LIN {X 0,Y 187.454,Z 298.954,A -85,B 0,C 180,E1 -22168.909,E2 -22168.909} C_VEL
LIN {X 0,Y 190.093,Z 301.065,A -85,B 0,C 180,E1 -22170.478,E2 -22170.478} C_VEL
LIN {X 0,Y 192.091,Z 304.274,A -85,B 0,C 180,E1 -22171.704,E2 -22171.704} C_VEL
LIN {X 0,Y 194.183,Z 306.294,A -85,B 0,C 180,E1 -22172.829,E2 -22172.829} C_VEL
LIN {X 0,Y 196.909,Z 310.048,A -85,B 0,C 180,E1 -22174.282,E2 -22174.282} C_VEL
LIN {X 0,Y 198.155,Z 311.601,A -85,B 0,C 180,E1 -22174.905,E2 -22174.905} C_VEL
LIN {X 0,Y 202.245,Z 317.198,A -85,B 0,C 180,E1 -22176.865,E2 -22176.865} C_VEL
LIN {X 0,Y 207.451,Z 324.554,A -85,B 0,C 180,E1 -22179.145,E2 -22179.145} C_VEL
LIN {X 0,Y 212.469,Z 332.432,A -85,B 0,C 180,E1 -22181.182,E2 -22181.182} C_VEL
LIN {X 0,Y 218.995,Z 345.187,A -85,B 0,C 180,E1 -22183.701,E2 -22183.701} C_VEL
LIN {X 0,Y 224.024,Z 356.545,A -85,B 0,C 180,E1 -22185.537,E2 -22185.537} C_VEL
LIN {X 0,Y 225.79,Z 360.908,A -85,B 0,C 180,E1 -22186.166,E2 -22186.166} C_VEL
LIN {X 0,Y 221.73,Z 427.354,A -85,B 0,C 180,E1 -22188.125,E2 -22188.125} C_VEL
LIN {X 0,Y 219.881,Z 441.769,A -85,B 0,C 180,E1 -22188.836,E2 -22188.836} C_VEL
LIN {X 0,Y 217.42,Z 455.664,A -85,B 0,C 180,E1 -22189.875,E2 -22189.875} C_VEL
LIN {X 0,Y 214.477,Z 468.601,A -85,B 0,C 180,E1 -22191.195,E2 -22191.195} C_VEL
LIN {X 0,Y 211.037,Z 481.143,A -85,B 0,C 180,E1 -22192.872,E2 -22192.872} C_VEL
LIN {X 0,Y 207.458,Z 492.576,A -85,B 0,C 180,E1 -22194.838,E2 -22194.838} C_VEL
LIN {X 0,Y 203.569,Z 503.074,A -85,B 0,C 180,E1 -22197.061,E2 -22197.061} C_VEL
LIN {X 0,Y 199.991,Z 511.877,A -85,B 0,C 180,E1 -22199.367,E2 -22199.367} C_VEL
LIN {X 0,Y 196.158,Z 520.748,A -85,B 0,C 180,E1 -22202.241,E2 -22202.241} C_VEL
LIN {X 0,Y 192.263,Z 529.243,A -85,B 0,C 180,E1 -22205.718,E2 -22205.718} C_VEL
LIN {X 0,Y 189.302,Z 536.081,A -85,B 0,C 180,E1 -22209.348,E2 -22209.348} C_VEL
LIN {X 0,Y 187.05,Z 540.801,A -85,B 0,C 180,E1 -22212.508,E2 -22212.508} C_VEL
LIN {X 0,Y 184.934,Z 545.689,A -85,B 0,C 180,E1 -22216.82,E2 -22216.82} C_VEL
LIN {X 0,Y 183.7,Z 549.087,A -85,B 0,C 180,E1 -22221.197,E2 -22221.197} C_VEL
LIN {X 0,Y 183.124,Z 551.102,A -85,B 0,C 180,E1 -22225.598,E2 -22225.598} C_VEL
LIN {X 0,Y 183.07,Z 551.787,A -85,B 0,C 180,E1 -22230,E2 -22230} C_VEL
LIN {X 0,Y 183.124,Z 551.153,A -85,B 0,C 180,E1 -22234.402,E2 -22234.402} C_VEL
LIN {X 0,Y 183.693,Z 549.184,A -85,B 0,C 180,E1 -22238.803,E2 -22238.803} C_VEL
LIN {X 0,Y 184.898,Z 545.833,A -85,B 0,C 180,E1 -22243.182,E2 -22243.182} C_VEL
LIN {X 0,Y 187.018,Z 540.999,A -85,B 0,C 180,E1 -22247.495,E2 -22247.495} C_VEL
LIN {X 0,Y 189.204,Z 536.332,A -85,B 0,C 180,E1 -22250.663,E2 -22250.663} C_VEL
LIN {X 0,Y 192.218,Z 529.549,A -85,B 0,C 180,E1 -22254.288,E2 -22254.288} C_VEL
LIN {X 0,Y 196.084,Z 521.119,A -85,B 0,C 180,E1 -22257.77,E2 -22257.77} C_VEL
LIN {X 0,Y 199.918,Z 512.321,A -85,B 0,C 180,E1 -22260.645,E2 -22260.645} C_VEL
LIN {X 0,Y 203.47,Z 503.606,A -85,B 0,C 180,E1 -22262.956,E2 -22262.956} C_VEL
LIN {X 0,Y 207.368,Z 493.216,A -85,B 0,C 180,E1 -22265.179,E2 -22265.179} C_VEL
LIN {X 0,Y 210.969,Z 481.914,A -85,B 0,C 180,E1 -22267.141,E2 -22267.141} C_VEL
LIN {X 0,Y 214.39,Z 469.557,A -85,B 0,C 180,E1 -22268.824,E2 -22268.824} C_VEL
LIN {X 0,Y 217.582,Z 455.768,A -85,B 0,C 180,E1 -22270.24,E2 -22270.24} C_VEL
LIN {X 0,Y 220.064,Z 441.904,A -85,B 0,C 180,E1 -22271.274,E2 -22271.274} C_VEL
LIN {X 0,Y 221.841,Z 427.094,A -85,B 0,C 180,E1 -22272.032,E2 -22272.032} C_VEL
LIN {X 0,Y 224.773,Z 380.963,A -85,B 0,C 180,E1 -22273.381,E2 -22273.381} C_VEL
LIN {X 0,Y 225.874,Z 360.793,A -85,B 0,C 180,E1 -22273.985,E2 -22273.985} C_VEL
LIN {X 0,Y 219.562,Z 346.139,A -85,B 0,C 180,E1 -22276.275,E2 -22276.275} C_VEL
LIN {X 0,Y 213.002,Z 333.315,A -85,B 0,C 180,E1 -22278.794,E2 -22278.794} C_VEL
LIN {X 0,Y 208.872,Z 326.562,A -85,B 0,C 180,E1 -22280.464,E2 -22280.464} C_VEL
LIN {X 0,Y 203.086,Z 318.318,A -85,B 0,C 180,E1 -22282.96,E2 -22282.96} C_VEL
LIN {X 0,Y 200.505,Z 314.745,A -85,B 0,C 180,E1 -22284.165,E2 -22284.165} C_VEL
LIN {X 0,Y 197.121,Z 310.237,A -85,B 0,C 180,E1 -22285.838,E2 -22285.838} C_VEL
LIN {X 0,Y 194.35,Z 306.597,A -85,B 0,C 180,E1 -22287.306,E2 -22287.306} C_VEL
LIN {X 0,Y 193.477,Z 305.537,A -85,B 0,C 180,E1 -22287.784,E2 -22287.784} C_VEL
LIN {X 0,Y 191.048,Z 302.837,A -85,B 0,C 180,E1 -22289.155,E2 -22289.155} C_VEL
LIN {X 0,Y 189.729,Z 300.609,A -85,B 0,C 180,E1 -22289.995,E2 -22289.995} C_VEL
LIN {X 0,Y 187.251,Z 298.716,A -85,B 0,C 180,E1 -22291.486,E2 -22291.486} C_VEL
LIN {X 0,Y 185.658,Z 295.648,A -85,B 0,C 180,E1 -22292.831,E2 -22292.831} C_VEL
LIN {X 0,Y 185.553,Z 295.014,A -85,B 0,C 180,E1 -22293.574,E2 -22293.574} C_VEL
LIN {X 0,Y 185.593,Z 294.976,A -85,B 0,C 180,E1 -22297.748,E2 -22297.748} C_VEL
LIN {X 0,Y 185.686,Z 294.979,A -85,B 0,C 180,E1 -22302.375,E2 -22302.375} C_VEL
LIN {X 0,Y 185.727,Z 294.959,A -85,B 0,C 180,E1 -22306.877,E2 -22306.877} C_VEL
LIN {X 0,Y 185.979,Z 294.915,A -85,B 0,C 180,E1 -22311.306,E2 -22311.306} C_VEL
LIN {X 0,Y 186.202,Z 294.886,A -85,B 0,C 180,E1 -22317.837,E2 -22317.837} C_VEL
LIN {X 0,Y 186.405,Z 294.881,A -85,B 0,C 180,E1 -22320,E2 -22320} C_VEL
LIN {X 0,Y 185.919,Z 294.922,A -85,B 0,C 180,E1 -22324.336,E2 -22324.336} C_VEL
LIN {X 0,Y 186.01,Z 294.921,A -85,B 0,C 180,E1 -22328.692,E2 -22328.692} C_VEL
LIN {X 0,Y 185.76,Z 294.97,A -85,B 0,C 180,E1 -22333.121,E2 -22333.121} C_VEL
LIN {X 0,Y 185.691,Z 294.975,A -85,B 0,C 180,E1 -22338.884,E2 -22338.884} C_VEL
LIN {X 0,Y 185.598,Z 294.99,A -85,B 0,C 180,E1 -22344.663,E2 -22344.663} C_VEL
LIN {X 0,Y 185.575,Z 295.249,A -85,B 0,C 180,E1 -22346.726,E2 -22346.726} C_VEL
LIN {X 0,Y 185.908,Z 296.393,A -85,B 0,C 180,E1 -22347.434,E2 -22347.434} C_VEL
LIN {X 0,Y 187.453,Z 298.923,A -85,B 0,C 180,E1 -22348.556,E2 -22348.556} C_VEL
LIN {X 0,Y 190.034,Z 300.979,A -85,B 0,C 180,E1 -22350.104,E2 -22350.104} C_VEL
LIN {X 0,Y 192.02,Z 304.151,A -85,B 0,C 180,E1 -22351.334,E2 -22351.334} C_VEL
LIN {X 0,Y 194.193,Z 306.346,A -85,B 0,C 180,E1 -22352.518,E2 -22352.518} C_VEL
LIN {X 0,Y 196.687,Z 309.82,A -85,B 0,C 180,E1 -22353.862,E2 -22353.862} C_VEL
LIN {X 0,Y 198.125,Z 311.496,A -85,B 0,C 180,E1 -22354.58,E2 -22354.58} C_VEL
LIN {X 0,Y 201.006,Z 315.29,A -85,B 0,C 180,E1 -22355.979,E2 -22355.979} C_VEL
LIN {X 0,Y 204.724,Z 320.809,A -85,B 0,C 180,E1 -22357.697,E2 -22357.697} C_VEL
LIN {X 0,Y 210.721,Z 330.915,A -85,B 0,C 180,E1 -22360.281,E2 -22360.281} C_VEL
LIN {X 0,Y 216.173,Z 341.306,A -85,B 0,C 180,E1 -22362.457,E2 -22362.457} C_VEL
LIN {X 0,Y 221.573,Z 352.961,A -85,B 0,C 180,E1 -22364.49,E2 -22364.49} C_VEL
LIN {X 0,Y 225.817,Z 363.464,A -85,B 0,C 180,E1 -22366.03,E2 -22366.03} C_VEL
LIN {X 0,Y 225.111,Z 375.8,A -85,B 0,C 180,E1 -22366.391,E2 -22366.391} C_VEL
LIN {X 0,Y 224.205,Z 381.65,A -85,B 0,C 180,E1 -22366.424,E2 -22366.424} C_VEL
LIN {X 0,Y 218.939,Z 400.687,A -85,B 0,C 180,E1 -22365.957,E2 -22365.957} C_VEL
LIN {X 0,Y 218.167,Z 406.528,A -85,B 0,C 180,E1 -22366.023,E2 -22366.023} C_VEL
LIN {X 0,Y 216.462,Z 431.011,A -85,B 0,C 180,E1 -22366.78,E2 -22366.78} C_VEL
LIN {X 0,Y 214.525,Z 445.259,A -85,B 0,C 180,E1 -22367.494,E2 -22367.494} C_VEL
LIN {X 0,Y 212.023,Z 458.486,A -85,B 0,C 180,E1 -22368.476,E2 -22368.476} C_VEL
LIN {X 0,Y 208.659,Z 472.362,A -85,B 0,C 180,E1 -22369.898,E2 -22369.898} C_VEL
LIN {X 0,Y 204.971,Z 484.787,A -85,B 0,C 180,E1 -22371.578,E2 -22371.578} C_VEL
LIN {X 0,Y 201.13,Z 496.148,A -85,B 0,C 180,E1 -22373.558,E2 -22373.558} C_VEL
LIN {X 0,Y 197.136,Z 506.591,A -85,B 0,C 180,E1 -22375.842,E2 -22375.842} C_VEL
LIN {X 0,Y 192.643,Z 516.981,A -85,B 0,C 180,E1 -22378.678,E2 -22378.678} C_VEL
LIN {X 0,Y 188.703,Z 525.554,A -85,B 0,C 180,E1 -22381.651,E2 -22381.651} C_VEL
LIN {X 0,Y 184.825,Z 533.759,A -85,B 0,C 180,E1 -22385.275,E2 -22385.275} C_VEL
LIN {X 0,Y 182.143,Z 539.511,A -85,B 0,C 180,E1 -22388.497,E2 -22388.497} C_VEL
LIN {X 0,Y 179.887,Z 544.219,A -85,B 0,C 180,E1 -22391.787,E2 -22391.787} C_VEL
LIN {X 0,Y 177.667,Z 549.098,A -85,B 0,C 180,E1 -22396.271,E2 -22396.271} C_VEL
LIN {X 0,Y 176.454,Z 552.491,A -85,B 0,C 180,E1 -22400.833,E2 -22400.833} C_VEL
LIN {X 0,Y 175.94,Z 554.495,A -85,B 0,C 180,E1 -22405.418,E2 -22405.418} C_VEL
LIN {X 0,Y 175.974,Z 555.154,A -85,B 0,C 180,E1 -22410,E2 -22410} C_VEL
LIN {X 0,Y 175.941,Z 554.475,A -85,B 0,C 180,E1 -22414.582,E2 -22414.582} C_VEL
LIN {X 0,Y 176.455,Z 552.452,A -85,B 0,C 180,E1 -22419.167,E2 -22419.167} C_VEL
LIN {X 0,Y 177.674,Z 549.038,A -85,B 0,C 180,E1 -22423.729,E2 -22423.729} C_VEL
LIN {X 0,Y 179.881,Z 544.132,A -85,B 0,C 180,E1 -22428.213,E2 -22428.213} C_VEL
LIN {X 0,Y 182.067,Z 539.401,A -85,B 0,C 180,E1 -22431.513,E2 -22431.513} C_VEL
LIN {X 0,Y 185.275,Z 532.543,A -85,B 0,C 180,E1 -22435.261,E2 -22435.261} C_VEL
LIN {X 0,Y 189.321,Z 524.034,A -85,B 0,C 180,E1 -22438.854,E2 -22438.854} C_VEL
LIN {X 0,Y 193.304,Z 515.153,A -85,B 0,C 180,E1 -22441.814,E2 -22441.814} C_VEL
LIN {X 0,Y 197.931,Z 504.398,A -85,B 0,C 180,E1 -22444.618,E2 -22444.618} C_VEL
LIN {X 0,Y 202.263,Z 492.687,A -85,B 0,C 180,E1 -22447.043,E2 -22447.043} C_VEL
LIN {X 0,Y 205.865,Z 481.583,A -85,B 0,C 180,E1 -22448.85,E2 -22448.85} C_VEL
LIN {X 0,Y 209.619,Z 468.366,A -85,B 0,C 180,E1 -22450.51,E2 -22450.51} C_VEL
LIN {X 0,Y 212.525,Z 455.61,A -85,B 0,C 180,E1 -22451.721,E2 -22451.721} C_VEL
LIN {X 0,Y 214.975,Z 441.144,A -85,B 0,C 180,E1 -22452.715,E2 -22452.715} C_VEL
LIN {X 0,Y 216.622,Z 427.426,A -85,B 0,C 180,E1 -22453.314,E2 -22453.314} C_VEL
LIN {X 0,Y 220.466,Z 366.13,A -85,B 0,C 180,E1 -22455.123,E2 -22455.123} C_VEL
LIN {X 0,Y 220.054,Z 364.331,A -85,B 0,C 180,E1 -22455.312,E2 -22455.312} C_VEL
LIN {X 0,Y 214.093,Z 350.156,A -85,B 0,C 180,E1 -22457.629,E2 -22457.629} C_VEL
LIN {X 0,Y 208.239,Z 338.338,A -85,B 0,C 180,E1 -22460.036,E2 -22460.036} C_VEL
LIN {X 0,Y 203.179,Z 329.197,A -85,B 0,C 180,E1 -22462.278,E2 -22462.278} C_VEL
LIN {X 0,Y 199.918,Z 323.95,A -85,B 0,C 180,E1 -22463.81,E2 -22463.81} C_VEL
LIN {X 0,Y 197.215,Z 320.172,A -85,B 0,C 180,E1 -22465.129,E2 -22465.129} C_VEL
LIN {X 0,Y 194.139,Z 315.981,A -85,B 0,C 180,E1 -22466.724,E2 -22466.724} C_VEL
LIN {X 0,Y 190.736,Z 311.521,A -85,B 0,C 180,E1 -22468.624,E2 -22468.624} C_VEL
LIN {X 0,Y 188.031,Z 308.074,A -85,B 0,C 180,E1 -22470.257,E2 -22470.257} C_VEL
LIN {X 0,Y 187.209,Z 306.892,A -85,B 0,C 180,E1 -22470.789,E2 -22470.789} C_VEL
LIN {X 0,Y 184.679,Z 304.486,A -85,B 0,C 180,E1 -22472.417,E2 -22472.417} C_VEL
LIN {X 0,Y 183.052,Z 301.671,A -85,B 0,C 180,E1 -22473.646,E2 -22473.646} C_VEL
LIN {X 0,Y 180.254,Z 299.692,A -85,B 0,C 180,E1 -22475.681,E2 -22475.681} C_VEL
LIN {X 0,Y 178.876,Z 297.326,A -85,B 0,C 180,E1 -22476.942,E2 -22476.942} C_VEL
LIN {X 0,Y 178.599,Z 296.163,A -85,B 0,C 180,E1 -22477.744,E2 -22477.744} C_VEL
LIN {X 0,Y 178.668,Z 295.839,A -85,B 0,C 180,E1 -22481.658,E2 -22481.658} C_VEL
LIN {X 0,Y 178.678,Z 295.853,A -85,B 0,C 180,E1 -22486.35,E2 -22486.35} C_VEL
LIN {X 0,Y 178.96,Z 295.795,A -85,B 0,C 180,E1 -22490.962,E2 -22490.962} C_VEL
LIN {X 0,Y 179.149,Z 295.774,A -85,B 0,C 180,E1 -22497.752,E2 -22497.752} C_VEL
LIN {X 0,Y 179.366,Z 295.757,A -85,B 0,C 180,E1 -22500,E2 -22500} C_VEL
LIN {X 0,Y 178.864,Z 295.814,A -85,B 0,C 180,E1 -22504.507,E2 -22504.507} C_VEL
LIN {X 0,Y 178.908,Z 295.795,A -85,B 0,C 180,E1 -22509.041,E2 -22509.041} C_VEL
LIN {X 0,Y 178.655,Z 295.835,A -85,B 0,C 180,E1 -22513.653,E2 -22513.653} C_VEL
LIN {X 0,Y 178.621,Z 295.845,A -85,B 0,C 180,E1 -22519.216,E2 -22519.216} C_VEL
LIN {X 0,Y 178.594,Z 296.138,A -85,B 0,C 180,E1 -22522.41,E2 -22522.41} C_VEL
LIN {X 0,Y 178.873,Z 297.38,A -85,B 0,C 180,E1 -22523.241,E2 -22523.241} C_VEL
LIN {X 0,Y 180.396,Z 299.812,A -85,B 0,C 180,E1 -22524.607,E2 -22524.607} C_VEL
LIN {X 0,Y 183.283,Z 301.984,A -85,B 0,C 180,E1 -22526.703,E2 -22526.703} C_VEL
LIN {X 0,Y 185.276,Z 305.274,A -85,B 0,C 180,E1 -22528.174,E2 -22528.174} C_VEL
LIN {X 0,Y 187.757,Z 307.536,A -85,B 0,C 180,E1 -22529.734,E2 -22529.734} C_VEL
LIN {X 0,Y 190.068,Z 310.88,A -85,B 0,C 180,E1 -22531.176,E2 -22531.176} C_VEL
LIN {X 0,Y 191.702,Z 312.631,A -85,B 0,C 180,E1 -22532.098,E2 -22532.098} C_VEL
LIN {X 0,Y 195.679,Z 318.017,A -85,B 0,C 180,E1 -22534.261,E2 -22534.261} C_VEL
LIN {X 0,Y 201.172,Z 325.585,A -85,B 0,C 180,E1 -22536.945,E2 -22536.945} C_VEL
LIN {X 0,Y 207.915,Z 335.897,A -85,B 0,C 180,E1 -22539.905,E2 -22539.905} C_VEL
LIN {X 0,Y 214.173,Z 348.148,A -85,B 0,C 180,E1 -22542.474,E2 -22542.474} C_VEL
LIN {X 0,Y 219.25,Z 359.843,A -85,B 0,C 180,E1 -22544.447,E2 -22544.447} C_VEL
LIN {X 0,Y 220.59,Z 363.064,A -85,B 0,C 180,E1 -22544.948,E2 -22544.948} C_VEL
LIN {X 0,Y 216.494,Z 427.614,A -85,B 0,C 180,E1 -22546.883,E2 -22546.883} C_VEL
LIN {X 0,Y 214.601,Z 441.845,A -85,B 0,C 180,E1 -22547.591,E2 -22547.591} C_VEL
LIN {X 0,Y 212.05,Z 455.738,A -85,B 0,C 180,E1 -22548.641,E2 -22548.641} C_VEL
LIN {X 0,Y 208.982,Z 468.673,A -85,B 0,C 180,E1 -22549.972,E2 -22549.972} C_VEL
LIN {X 0,Y 205.408,Z 481.215,A -85,B 0,C 180,E1 -22551.674,E2 -22551.674} C_VEL
LIN {X 0,Y 201.696,Z 492.646,A -85,B 0,C 180,E1 -22553.676,E2 -22553.676} C_VEL
LIN {X 0,Y 197.645,Z 503.144,A -85,B 0,C 180,E1 -22555.942,E2 -22555.942} C_VEL
LIN {X 0,Y 193.9,Z 511.946,A -85,B 0,C 180,E1 -22558.295,E2 -22558.295} C_VEL
LIN {X 0,Y 189.902,Z 520.817,A -85,B 0,C 180,E1 -22561.243,E2 -22561.243} C_VEL
LIN {X 0,Y 185.778,Z 529.312,A -85,B 0,C 180,E1 -22564.812,E2 -22564.812} C_VEL
LIN {X 0,Y 182.632,Z 536.15,A -85,B 0,C 180,E1 -22568.557,E2 -22568.557} C_VEL
LIN {X 0,Y 180.284,Z 540.869,A -85,B 0,C 180,E1 -22571.829,E2 -22571.829} C_VEL
LIN {X 0,Y 178.001,Z 545.757,A -85,B 0,C 180,E1 -22576.297,E2 -22576.297} C_VEL
LIN {X 0,Y 176.66,Z 549.155,A -85,B 0,C 180,E1 -22580.844,E2 -22580.844} C_VEL
LIN {X 0,Y 176.035,Z 551.169,A -85,B 0,C 180,E1 -22585.42,E2 -22585.42} C_VEL
LIN {X 0,Y 175.983,Z 551.853,A -85,B 0,C 180,E1 -22590,E2 -22590} C_VEL
LIN {X 0,Y 176.035,Z 551.22,A -85,B 0,C 180,E1 -22594.58,E2 -22594.58} C_VEL
LIN {X 0,Y 176.317,Z 550.404,A -85,B 0,C 180,E1 -22596.868,E2 -22596.868} C_VEL
LIN {X 0,Y 177.208,Z 547.752,A -85,B 0,C 180,E1 -22601.437,E2 -22601.437} C_VEL
LIN {X 0,Y 178.93,Z 543.677,A -85,B 0,C 180,E1 -22605.958,E2 -22605.958} C_VEL
LIN {X 0,Y 181.764,Z 538.044,A -85,B 0,C 180,E1 -22610.364,E2 -22610.364} C_VEL
LIN {X 0,Y 184.427,Z 532.24,A -85,B 0,C 180,E1 -22613.854,E2 -22613.854} C_VEL
LIN {X 0,Y 187.954,Z 525.009,A -85,B 0,C 180,E1 -22617.261,E2 -22617.261} C_VEL
LIN {X 0,Y 191.749,Z 516.99,A -85,B 0,C 180,E1 -22620.262,E2 -22620.262} C_VEL
LIN {X 0,Y 196.008,Z 507.318,A -85,B 0,C 180,E1 -22623.147,E2 -22623.147} C_VEL
LIN {X 0,Y 200.357,Z 496.582,A -85,B 0,C 180,E1 -22625.672,E2 -22625.672} C_VEL
LIN {X 0,Y 204.271,Z 485.325,A -85,B 0,C 180,E1 -22627.795,E2 -22627.795} C_VEL
LIN {X 0,Y 207.989,Z 472.982,A -85,B 0,C 180,E1 -22629.626,E2 -22629.626} C_VEL
LIN {X 0,Y 211.487,Z 459.199,A -85,B 0,C 180,E1 -22631.176,E2 -22631.176} C_VEL
LIN {X 0,Y 214.288,Z 445.008,A -85,B 0,C 180,E1 -22632.326,E2 -22632.326} C_VEL
LIN {X 0,Y 216.219,Z 430.925,A -85,B 0,C 180,E1 -22633.124,E2 -22633.124} C_VEL
LIN {X 0,Y 217.647,Z 413.223,A -85,B 0,C 180,E1 -22633.722,E2 -22633.722} C_VEL
LIN {X 0,Y 220.74,Z 363.261,A -85,B 0,C 180,E1 -22635.175,E2 -22635.175} C_VEL
LIN {X 0,Y 214.832,Z 349.379,A -85,B 0,C 180,E1 -22637.455,E2 -22637.455} C_VEL
LIN {X 0,Y 208.881,Z 337.599,A -85,B 0,C 180,E1 -22639.88,E2 -22639.88} C_VEL
LIN {X 0,Y 204.45,Z 330.464,A -85,B 0,C 180,E1 -22641.775,E2 -22641.775} C_VEL
LIN {X 0,Y 199.739,Z 323.617,A -85,B 0,C 180,E1 -22643.936,E2 -22643.936} C_VEL
LIN {X 0,Y 197.014,Z 319.876,A -85,B 0,C 180,E1 -22645.274,E2 -22645.274} C_VEL
LIN {X 0,Y 194.243,Z 316.045,A -85,B 0,C 180,E1 -22646.726,E2 -22646.726} C_VEL
LIN {X 0,Y 190.913,Z 311.665,A -85,B 0,C 180,E1 -22648.592,E2 -22648.592} C_VEL
LIN {X 0,Y 188.243,Z 308.406,A -85,B 0,C 180,E1 -22650.197,E2 -22650.197} C_VEL
LIN {X 0,Y 187.316,Z 306.978,A -85,B 0,C 180,E1 -22650.807,E2 -22650.807} C_VEL
LIN {X 0,Y 184.793,Z 304.619,A -85,B 0,C 180,E1 -22652.435,E2 -22652.435} C_VEL
LIN {X 0,Y 183.002,Z 301.629,A -85,B 0,C 180,E1 -22653.791,E2 -22653.791} C_VEL
LIN {X 0,Y 180.275,Z 299.7,A -85,B 0,C 180,E1 -22655.797,E2 -22655.797} C_VEL
LIN {X 0,Y 178.869,Z 297.339,A -85,B 0,C 180,E1 -22657.093,E2 -22657.093} C_VEL
LIN {X 0,Y 178.6,Z 296.144,A -85,B 0,C 180,E1 -22657.896,E2 -22657.896} C_VEL
LIN {X 0,Y 178.647,Z 295.852,A -85,B 0,C 180,E1 -22661.656,E2 -22661.656} C_VEL
LIN {X 0,Y 178.654,Z 295.834,A -85,B 0,C 180,E1 -22666.347,E2 -22666.347} C_VEL
LIN {X 0,Y 178.908,Z 295.795,A -85,B 0,C 180,E1 -22670.959,E2 -22670.959} C_VEL
LIN {X 0,Y 178.863,Z 295.815,A -85,B 0,C 180,E1 -22675.493,E2 -22675.493} C_VEL
LIN {X 0,Y 179.368,Z 295.756,A -85,B 0,C 180,E1 -22680,E2 -22680} C_VEL
LIN {X 0,Y 178.867,Z 295.8,A -85,B 0,C 180,E1 -22684.507,E2 -22684.507} C_VEL
LIN {X 0,Y 178.959,Z 295.795,A -85,B 0,C 180,E1 -22689.038,E2 -22689.038} C_VEL
LIN {X 0,Y 178.678,Z 295.853,A -85,B 0,C 180,E1 -22693.65,E2 -22693.65} C_VEL
LIN {X 0,Y 178.635,Z 295.858,A -85,B 0,C 180,E1 -22699.23,E2 -22699.23} C_VEL
LIN {X 0,Y 178.58,Z 296.111,A -85,B 0,C 180,E1 -22701.954,E2 -22701.954} C_VEL
LIN {X 0,Y 178.881,Z 297.333,A -85,B 0,C 180,E1 -22702.828,E2 -22702.828} C_VEL
LIN {X 0,Y 180.264,Z 299.713,A -85,B 0,C 180,E1 -22704.109,E2 -22704.109} C_VEL
LIN {X 0,Y 183.272,Z 301.941,A -85,B 0,C 180,E1 -22706.32,E2 -22706.32} C_VEL
LIN {X 0,Y 185.132,Z 305.07,A -85,B 0,C 180,E1 -22707.716,E2 -22707.716} C_VEL
LIN {X 0,Y 187.706,Z 307.47,A -85,B 0,C 180,E1 -22709.357,E2 -22709.357} C_VEL
LIN {X 0,Y 190.205,Z 310.974,A -85,B 0,C 180,E1 -22710.919,E2 -22710.919} C_VEL
LIN {X 0,Y 191.745,Z 312.736,A -85,B 0,C 180,E1 -22711.801,E2 -22711.801} C_VEL
LIN {X 0,Y 194.803,Z 316.628,A -85,B 0,C 180,E1 -22713.476,E2 -22713.476} C_VEL
LIN {X 0,Y 200.959,Z 325.382,A -85,B 0,C 180,E1 -22716.557,E2 -22716.557} C_VEL
LIN {X 0,Y 207.456,Z 336.652,A -85,B 0,C 180,E1 -22719.513,E2 -22719.513} C_VEL
LIN {X 0,Y 213.162,Z 347.977,A -85,B 0,C 180,E1 -22721.897,E2 -22721.897} C_VEL
LIN {X 0,Y 218.609,Z 360.499,A -85,B 0,C 180,E1 -22724.044,E2 -22724.044} C_VEL
LIN {X 0,Y 220.584,Z 365.634,A -85,B 0,C 180,E1 -22724.804,E2 -22724.804} C_VEL
LIN {X 0,Y 218.167,Z 406.528,A -85,B 0,C 180,E1 -22726.023,E2 -22726.023} C_VEL
LIN {X 0,Y 217.388,Z 412.381,A -85,B 0,C 180,E1 -22726.076,E2 -22726.076} C_VEL
LIN {X 0,Y 211.798,Z 431.345,A -85,B 0,C 180,E1 -22725.588,E2 -22725.588} C_VEL
LIN {X 0,Y 210.597,Z 437.105,A -85,B 0,C 180,E1 -22725.73,E2 -22725.73} C_VEL
LIN {X 0,Y 208.279,Z 451.016,A -85,B 0,C 180,E1 -22726.568,E2 -22726.568} C_VEL
LIN {X 0,Y 205.263,Z 464.84,A -85,B 0,C 180,E1 -22727.784,E2 -22727.784} C_VEL
LIN {X 0,Y 201.791,Z 477.277,A -85,B 0,C 180,E1 -22729.231,E2 -22729.231} C_VEL
LIN {X 0,Y 197.969,Z 489.006,A -85,B 0,C 180,E1 -22731.007,E2 -22731.007} C_VEL
LIN {X 0,Y 193.566,Z 501.01,A -85,B 0,C 180,E1 -22733.358,E2 -22733.358} C_VEL
LIN {X 0,Y 188.876,Z 511.979,A -85,B 0,C 180,E1 -22736.073,E2 -22736.073} C_VEL
LIN {X 0,Y 184.516,Z 521.403,A -85,B 0,C 180,E1 -22739.057,E2 -22739.057} C_VEL
LIN {X 0,Y 179.982,Z 530.376,A -85,B 0,C 180,E1 -22742.69,E2 -22742.69} C_VEL
LIN {X 0,Y 176.297,Z 537.631,A -85,B 0,C 180,E1 -22746.507,E2 -22746.507} C_VEL
LIN {X 0,Y 173.841,Z 542.718,A -85,B 0,C 180,E1 -22749.902,E2 -22749.902} C_VEL
LIN {X 0,Y 171.181,Z 547.964,A -85,B 0,C 180,E1 -22754.523,E2 -22754.523} C_VEL
LIN {X 0,Y 169.977,Z 550.906,A -85,B 0,C 180,E1 -22758.069,E2 -22758.069} C_VEL
LIN {X 0,Y 169.071,Z 553.597,A -85,B 0,C 180,E1 -22762.837,E2 -22762.837} C_VEL
LIN {X 0,Y 168.782,Z 554.925,A -85,B 0,C 180,E1 -22767.614,E2 -22767.614} C_VEL
LIN {X 0,Y 168.872,Z 555.088,A -85,B 0,C 180,E1 -22770,E2 -22770} C_VEL
LIN {X 0,Y 168.859,Z 554.408,A -85,B 0,C 180,E1 -22774.775,E2 -22774.775} C_VEL
LIN {X 0,Y 169.41,Z 552.385,A -85,B 0,C 180,E1 -22779.552,E2 -22779.552} C_VEL
LIN {X 0,Y 170.727,Z 548.97,A -85,B 0,C 180,E1 -22784.299,E2 -22784.299} C_VEL
LIN {X 0,Y 173.121,Z 544.064,A -85,B 0,C 180,E1 -22788.951,E2 -22788.951} C_VEL
LIN {X 0,Y 176.171,Z 537.634,A -85,B 0,C 180,E1 -22793.431,E2 -22793.431} C_VEL
LIN {X 0,Y 179.976,Z 530.239,A -85,B 0,C 180,E1 -22797.311,E2 -22797.311} C_VEL
LIN {X 0,Y 184.48,Z 521.218,A -85,B 0,C 180,E1 -22800.95,E2 -22800.95} C_VEL
LIN {X 0,Y 188.861,Z 511.756,A -85,B 0,C 180,E1 -22803.93,E2 -22803.93} C_VEL
LIN {X 0,Y 193.589,Z 500.7,A -85,B 0,C 180,E1 -22806.65,E2 -22806.65} C_VEL
LIN {X 0,Y 197.957,Z 488.68,A -85,B 0,C 180,E1 -22808.997,E2 -22808.997} C_VEL
LIN {X 0,Y 201.812,Z 476.878,A -85,B 0,C 180,E1 -22810.764,E2 -22810.764} C_VEL
LIN {X 0,Y 205.249,Z 464.325,A -85,B 0,C 180,E1 -22812.219,E2 -22812.219} C_VEL
LIN {X 0,Y 208.301,Z 450.336,A -85,B 0,C 180,E1 -22813.427,E2 -22813.427} C_VEL
LIN {X 0,Y 210.506,Z 436.486,A -85,B 0,C 180,E1 -22814.264,E2 -22814.264} C_VEL
LIN {X 0,Y 211.853,Z 422.899,A -85,B 0,C 180,E1 -22814.788,E2 -22814.788} C_VEL
LIN {X 0,Y 215.36,Z 367.704,A -85,B 0,C 180,E1 -22816.425,E2 -22816.425} C_VEL
LIN {X 0,Y 210.087,Z 354.818,A -85,B 0,C 180,E1 -22818.6,E2 -22818.6} C_VEL
LIN {X 0,Y 204.927,Z 344.08,A -85,B 0,C 180,E1 -22820.838,E2 -22820.838} C_VEL
LIN {X 0,Y 200.599,Z 335.968,A -85,B 0,C 180,E1 -22822.844,E2 -22822.844} C_VEL
LIN {X 0,Y 196.741,Z 329.427,A -85,B 0,C 180,E1 -22824.751,E2 -22824.751} C_VEL
LIN {X 0,Y 193.799,Z 325.242,A -85,B 0,C 180,E1 -22826.269,E2 -22826.269} C_VEL
LIN {X 0,Y 191.171,Z 321.626,A -85,B 0,C 180,E1 -22827.711,E2 -22827.711} C_VEL
LIN {X 0,Y 188.26,Z 317.643,A -85,B 0,C 180,E1 -22829.427,E2 -22829.427} C_VEL
LIN {X 0,Y 185.429,Z 313.875,A -85,B 0,C 180,E1 -22831.231,E2 -22831.231} C_VEL
LIN {X 0,Y 182.117,Z 310.181,A -85,B 0,C 180,E1 -22833.5,E2 -22833.5} C_VEL
LIN {X 0,Y 180.888,Z 308.177,A -85,B 0,C 180,E1 -22834.468,E2 -22834.468} C_VEL
LIN {X 0,Y 178.197,Z 305.913,A -85,B 0,C 180,E1 -22836.559,E2 -22836.559} C_VEL
LIN {X 0,Y 176.589,Z 303.022,A -85,B 0,C 180,E1 -22838.092,E2 -22838.092} C_VEL
LIN {X 0,Y 173.22,Z 300.417,A -85,B 0,C 180,E1 -22841.367,E2 -22841.367} C_VEL
LIN {X 0,Y 171.707,Z 297.39,A -85,B 0,C 180,E1 -22843.657,E2 -22843.657} C_VEL
LIN {X 0,Y 171.579,Z 296.782,A -85,B 0,C 180,E1 -22845.167,E2 -22845.167} C_VEL
LIN {X 0,Y 171.888,Z 296.672,A -85,B 0,C 180,E1 -22850.587,E2 -22850.587} C_VEL
LIN {X 0,Y 171.817,Z 296.678,A -85,B 0,C 180,E1 -22855.308,E2 -22855.308} C_VEL
LIN {X 0,Y 172.329,Z 296.632,A -85,B 0,C 180,E1 -22860,E2 -22860} C_VEL
LIN {X 0,Y 171.812,Z 296.694,A -85,B 0,C 180,E1 -22864.693,E2 -22864.693} C_VEL
LIN {X 0,Y 171.845,Z 296.675,A -85,B 0,C 180,E1 -22869.415,E2 -22869.415} C_VEL
LIN {X 0,Y 171.631,Z 296.996,A -85,B 0,C 180,E1 -22875.893,E2 -22875.893} C_VEL
LIN {X 0,Y 171.848,Z 298.02,A -85,B 0,C 180,E1 -22877.018,E2 -22877.018} C_VEL
LIN {X 0,Y 173.447,Z 300.705,A -85,B 0,C 180,E1 -22879.066,E2 -22879.066} C_VEL
LIN {X 0,Y 176.565,Z 303.016,A -85,B 0,C 180,E1 -22882.065,E2 -22882.065} C_VEL
LIN {X 0,Y 178.234,Z 305.929,A -85,B 0,C 180,E1 -22883.647,E2 -22883.647} C_VEL
LIN {X 0,Y 180.772,Z 308.119,A -85,B 0,C 180,E1 -22885.627,E2 -22885.627} C_VEL
LIN {X 0,Y 181.762,Z 309.589,A -85,B 0,C 180,E1 -22886.402,E2 -22886.402} C_VEL
LIN {X 0,Y 184.113,Z 312.603,A -85,B 0,C 180,E1 -22888.091,E2 -22888.091} C_VEL
LIN {X 0,Y 185.467,Z 313.931,A -85,B 0,C 180,E1 -22888.972,E2 -22888.972} C_VEL
LIN {X 0,Y 188.229,Z 317.641,A -85,B 0,C 180,E1 -22890.734,E2 -22890.734} C_VEL
LIN {X 0,Y 189.641,Z 319.484,A -85,B 0,C 180,E1 -22891.578,E2 -22891.578} C_VEL
LIN {X 0,Y 193.379,Z 324.627,A -85,B 0,C 180,E1 -22893.682,E2 -22893.682} C_VEL
LIN {X 0,Y 198.067,Z 331.213,A -85,B 0,C 180,E1 -22896.072,E2 -22896.072} C_VEL
LIN {X 0,Y 204.575,Z 341.496,A -85,B 0,C 180,E1 -22899.077,E2 -22899.077} C_VEL
LIN {X 0,Y 210.282,Z 353.017,A -85,B 0,C 180,E1 -22901.546,E2 -22901.546} C_VEL
LIN {X 0,Y 215.25,Z 364.846,A -85,B 0,C 180,E1 -22903.586,E2 -22903.586} C_VEL
LIN {X 0,Y 215.492,Z 365.42,A -85,B 0,C 180,E1 -22903.681,E2 -22903.681} C_VEL
LIN {X 0,Y 211.439,Z 426.97,A -85,B 0,C 180,E1 -22905.534,E2 -22905.534} C_VEL
LIN {X 0,Y 209.556,Z 441.16,A -85,B 0,C 180,E1 -22906.235,E2 -22906.235} C_VEL
LIN {X 0,Y 207.03,Z 454.683,A -85,B 0,C 180,E1 -22907.241,E2 -22907.241} C_VEL
LIN {X 0,Y 204.087,Z 466.98,A -85,B 0,C 180,E1 -22908.48,E2 -22908.48} C_VEL
LIN {X 0,Y 200.348,Z 479.862,A -85,B 0,C 180,E1 -22910.195,E2 -22910.195} C_VEL
LIN {X 0,Y 196.696,Z 490.913,A -85,B 0,C 180,E1 -22912.101,E2 -22912.101} C_VEL
LIN {X 0,Y 192.637,Z 501.265,A -85,B 0,C 180,E1 -22914.287,E2 -22914.287} C_VEL
LIN {X 0,Y 188.588,Z 510.392,A -85,B 0,C 180,E1 -22916.656,E2 -22916.656} C_VEL
LIN {X 0,Y 184.349,Z 519.535,A -85,B 0,C 180,E1 -22919.66,E2 -22919.66} C_VEL
LIN {X 0,Y 179.904,Z 528.268,A -85,B 0,C 180,E1 -22923.305,E2 -22923.305} C_VEL
LIN {X 0,Y 176.868,Z 534.415,A -85,B 0,C 180,E1 -22926.587,E2 -22926.587} C_VEL
LIN {X 0,Y 174.322,Z 539.498,A -85,B 0,C 180,E1 -22929.96,E2 -22929.96} C_VEL
LIN {X 0,Y 171.58,Z 544.764,A -85,B 0,C 180,E1 -22934.559,E2 -22934.559} C_VEL
LIN {X 0,Y 170.264,Z 547.702,A -85,B 0,C 180,E1 -22938.089,E2 -22938.089} C_VEL
LIN {X 0,Y 169.259,Z 550.397,A -85,B 0,C 180,E1 -22942.844,E2 -22942.844} C_VEL
LIN {X 0,Y 168.859,Z 551.743,A -85,B 0,C 180,E1 -22947.615,E2 -22947.615} C_VEL
LIN {X 0,Y 168.882,Z 551.92,A -85,B 0,C 180,E1 -22950,E2 -22950} C_VEL
LIN {X 0,Y 168.952,Z 551.286,A -85,B 0,C 180,E1 -22954.772,E2 -22954.772} C_VEL
LIN {X 0,Y 169.634,Z 549.316,A -85,B 0,C 180,E1 -22959.539,E2 -22959.539} C_VEL
LIN {X 0,Y 171.063,Z 545.965,A -85,B 0,C 180,E1 -22964.27,E2 -22964.27} C_VEL
LIN {X 0,Y 173.479,Z 541.13,A -85,B 0,C 180,E1 -22968.91,E2 -22968.91} C_VEL
LIN {X 0,Y 175.9,Z 536.463,A -85,B 0,C 180,E1 -22972.306,E2 -22972.306} C_VEL
LIN {X 0,Y 179.322,Z 529.679,A -85,B 0,C 180,E1 -22976.161,E2 -22976.161} C_VEL
LIN {X 0,Y 182.937,Z 522.598,A -85,B 0,C 180,E1 -22979.328,E2 -22979.328} C_VEL
LIN {X 0,Y 187.078,Z 514.071,A -85,B 0,C 180,E1 -22982.365,E2 -22982.365} C_VEL
LIN {X 0,Y 190.881,Z 505.603,A -85,B 0,C 180,E1 -22984.797,E2 -22984.797} C_VEL
LIN {X 0,Y 195.459,Z 494.501,A -85,B 0,C 180,E1 -22987.355,E2 -22987.355} C_VEL
LIN {X 0,Y 199.817,Z 482.038,A -85,B 0,C 180,E1 -22989.604,E2 -22989.604} C_VEL
LIN {X 0,Y 203.547,Z 469.678,A -85,B 0,C 180,E1 -22991.325,E2 -22991.325} C_VEL
LIN {X 0,Y 206.97,Z 455.887,A -85,B 0,C 180,E1 -22992.775,E2 -22992.775} C_VEL
LIN {X 0,Y 209.505,Z 442.779,A -85,B 0,C 180,E1 -22993.778,E2 -22993.778} C_VEL
LIN {X 0,Y 211.3,Z 428.993,A -85,B 0,C 180,E1 -22994.531,E2 -22994.531} C_VEL
LIN {X 0,Y 213.24,Z 404.576,A -85,B 0,C 180,E1 -22995.271,E2 -22995.271} C_VEL
LIN {X 0,Y 215.582,Z 365.358,A -85,B 0,C 180,E1 -22996.474,E2 -22996.474} C_VEL
LIN {X 0,Y 210.401,Z 353.11,A -85,B 0,C 180,E1 -22998.599,E2 -22998.599} C_VEL
LIN {X 0,Y 204.377,Z 340.998,A -85,B 0,C 180,E1 -23001.217,E2 -23001.217} C_VEL
LIN {X 0,Y 198.595,Z 332.032,A -85,B 0,C 180,E1 -23003.882,E2 -23003.882} C_VEL
LIN {X 0,Y 194.195,Z 325.729,A -85,B 0,C 180,E1 -23006.112,E2 -23006.112} C_VEL
LIN {X 0,Y 191.149,Z 321.539,A -85,B 0,C 180,E1 -23007.788,E2 -23007.788} C_VEL
LIN {X 0,Y 188.379,Z 317.774,A -85,B 0,C 180,E1 -23009.428,E2 -23009.428} C_VEL
LIN {X 0,Y 185.589,Z 314.099,A -85,B 0,C 180,E1 -23011.211,E2 -23011.211} C_VEL
LIN {X 0,Y 184.444,Z 312.886,A -85,B 0,C 180,E1 -23011.964,E2 -23011.964} C_VEL
LIN {X 0,Y 181.822,Z 309.701,A -85,B 0,C 180,E1 -23013.839,E2 -23013.839} C_VEL
LIN {X 0,Y 180.941,Z 308.176,A -85,B 0,C 180,E1 -23014.552,E2 -23014.552} C_VEL
LIN {X 0,Y 178.233,Z 305.971,A -85,B 0,C 180,E1 -23016.671,E2 -23016.671} C_VEL
LIN {X 0,Y 176.471,Z 302.759,A -85,B 0,C 180,E1 -23018.384,E2 -23018.384} C_VEL
LIN {X 0,Y 173.522,Z 300.779,A -85,B 0,C 180,E1 -23021.247,E2 -23021.247} C_VEL
LIN {X 0,Y 171.876,Z 298.136,A -85,B 0,C 180,E1 -23023.367,E2 -23023.367} C_VEL
LIN {X 0,Y 171.637,Z 297.178,A -85,B 0,C 180,E1 -23024.26,E2 -23024.26} C_VEL
LIN {X 0,Y 171.578,Z 296.766,A -85,B 0,C 180,E1 -23025.773,E2 -23025.773} C_VEL
LIN {X 0,Y 171.844,Z 296.676,A -85,B 0,C 180,E1 -23030.584,E2 -23030.584} C_VEL
LIN {X 0,Y 171.812,Z 296.695,A -85,B 0,C 180,E1 -23035.307,E2 -23035.307} C_VEL
LIN {X 0,Y 172.331,Z 296.632,A -85,B 0,C 180,E1 -23040,E2 -23040} C_VEL
LIN {X 0,Y 171.816,Z 296.678,A -85,B 0,C 180,E1 -23044.692,E2 -23044.692} C_VEL
LIN {X 0,Y 171.888,Z 296.672,A -85,B 0,C 180,E1 -23049.413,E2 -23049.413} C_VEL
LIN {X 0,Y 171.593,Z 296.9,A -85,B 0,C 180,E1 -23055.135,E2 -23055.135} C_VEL
LIN {X 0,Y 171.794,Z 297.772,A -85,B 0,C 180,E1 -23056.335,E2 -23056.335} C_VEL
LIN {X 0,Y 173.226,Z 300.403,A -85,B 0,C 180,E1 -23058.326,E2 -23058.326} C_VEL
LIN {X 0,Y 175.673,Z 302.368,A -85,B 0,C 180,E1 -23060.817,E2 -23060.817} C_VEL
LIN {X 0,Y 176.612,Z 303.036,A -85,B 0,C 180,E1 -23061.674,E2 -23061.674} C_VEL
LIN {X 0,Y 178.32,Z 306.081,A -85,B 0,C 180,E1 -23063.318,E2 -23063.318} C_VEL
LIN {X 0,Y 181.294,Z 308.724,A -85,B 0,C 180,E1 -23065.644,E2 -23065.644} C_VEL
LIN {X 0,Y 183.559,Z 312.007,A -85,B 0,C 180,E1 -23067.351,E2 -23067.351} C_VEL
LIN {X 0,Y 185.473,Z 313.931,A -85,B 0,C 180,E1 -23068.623,E2 -23068.623} C_VEL
LIN {X 0,Y 188.366,Z 317.753,A -85,B 0,C 180,E1 -23070.476,E2 -23070.476} C_VEL
LIN {X 0,Y 192.85,Z 323.835,A -85,B 0,C 180,E1 -23073.074,E2 -23073.074} C_VEL
LIN {X 0,Y 197.756,Z 330.784,A -85,B 0,C 180,E1 -23075.62,E2 -23075.62} C_VEL
LIN {X 0,Y 204.092,Z 342.14,A -85,B 0,C 180,E1 -23078.659,E2 -23078.659} C_VEL
LIN {X 0,Y 210.109,Z 354.553,A -85,B 0,C 180,E1 -23081.296,E2 -23081.296} C_VEL
LIN {X 0,Y 215.492,Z 367.807,A -85,B 0,C 180,E1 -23083.529,E2 -23083.529} C_VEL
LIN {X 0,Y 211.439,Z 430.217,A -85,B 0,C 180,E1 -23085.433,E2 -23085.433} C_VEL
LIN {X 0,Y 210.597,Z 437.105,A -85,B 0,C 180,E1 -23085.73,E2 -23085.73} C_VEL
LIN {X 0,Y 209.792,Z 440.923,A -85,B 0,C 180,E1 -23085.865,E2 -23085.865} C_VEL
LIN {X 0,Y 207.133,Z 448.366,A -85,B 0,C 180,E1 -23085.944,E2 -23085.944} C_VEL
LIN {X 0,Y 201.456,Z 461.038,A -85,B 0,C 180,E1 -23086.167,E2 -23086.167} C_VEL
LIN {X 0,Y 199.613,Z 466.423,A -85,B 0,C 180,E1 -23086.583,E2 -23086.583} C_VEL
LIN {X 0,Y 195.962,Z 478.798,A -85,B 0,C 180,E1 -23088.091,E2 -23088.091} C_VEL
LIN {X 0,Y 191.667,Z 491.27,A -85,B 0,C 180,E1 -23090.084,E2 -23090.084} C_VEL
LIN {X 0,Y 187.098,Z 502.966,A -85,B 0,C 180,E1 -23092.524,E2 -23092.524} C_VEL
LIN {X 0,Y 182.201,Z 513.595,A -85,B 0,C 180,E1 -23095.324,E2 -23095.324} C_VEL
LIN {X 0,Y 177.712,Z 522.714,A -85,B 0,C 180,E1 -23098.4,E2 -23098.4} C_VEL
LIN {X 0,Y 173.064,Z 531.429,A -85,B 0,C 180,E1 -23102.161,E2 -23102.161} C_VEL
LIN {X 0,Y 169.601,Z 537.863,A -85,B 0,C 180,E1 -23105.734,E2 -23105.734} C_VEL
LIN {X 0,Y 166.382,Z 544.087,A -85,B 0,C 180,E1 -23110.25,E2 -23110.25} C_VEL
LIN {X 0,Y 163.793,Z 548.965,A -85,B 0,C 180,E1 -23115.082,E2 -23115.082} C_VEL
LIN {X 0,Y 162.388,Z 552.358,A -85,B 0,C 180,E1 -23120.031,E2 -23120.031} C_VEL
LIN {X 0,Y 161.766,Z 554.363,A -85,B 0,C 180,E1 -23125.016,E2 -23125.016} C_VEL
LIN {X 0,Y 161.772,Z 555.021,A -85,B 0,C 180,E1 -23130,E2 -23130} C_VEL
LIN {X 0,Y 161.766,Z 554.341,A -85,B 0,C 180,E1 -23134.985,E2 -23134.985} C_VEL
LIN {X 0,Y 162.389,Z 552.317,A -85,B 0,C 180,E1 -23139.969,E2 -23139.969} C_VEL
LIN {X 0,Y 163.803,Z 548.902,A -85,B 0,C 180,E1 -23144.917,E2 -23144.917} C_VEL
LIN {X 0,Y 166.37,Z 543.996,A -85,B 0,C 180,E1 -23149.751,E2 -23149.751} C_VEL
LIN {X 0,Y 169.417,Z 537.978,A -85,B 0,C 180,E1 -23154.128,E2 -23154.128} C_VEL
LIN {X 0,Y 173.058,Z 531.288,A -85,B 0,C 180,E1 -23157.841,E2 -23157.841} C_VEL
LIN {X 0,Y 177.688,Z 522.54,A -85,B 0,C 180,E1 -23161.605,E2 -23161.605} C_VEL
LIN {X 0,Y 182.189,Z 513.386,A -85,B 0,C 180,E1 -23164.679,E2 -23164.679} C_VEL
LIN {X 0,Y 187.118,Z 502.686,A -85,B 0,C 180,E1 -23167.479,E2 -23167.479} C_VEL
LIN {X 0,Y 191.635,Z 490.935,A -85,B 0,C 180,E1 -23169.925,E2 -23169.925} C_VEL
LIN {X 0,Y 195.98,Z 478.389,A -85,B 0,C 180,E1 -23171.905,E2 -23171.905} C_VEL
LIN {X 0,Y 199.545,Z 466.242,A -85,B 0,C 180,E1 -23173.376,E2 -23173.376} C_VEL
LIN {X 0,Y 202.689,Z 452.864,A -85,B 0,C 180,E1 -23174.598,E2 -23174.598} C_VEL
LIN {X 0,Y 205.036,Z 439.158,A -85,B 0,C 180,E1 -23175.51,E2 -23175.51} C_VEL
LIN {X 0,Y 206.609,Z 426.273,A -85,B 0,C 180,E1 -23176.05,E2 -23176.05} C_VEL
LIN {X 0,Y 210.375,Z 369.956,A -85,B 0,C 180,E1 -23177.754,E2 -23177.754} C_VEL
LIN {X 0,Y 205.186,Z 357.254,A -85,B 0,C 180,E1 -23180.042,E2 -23180.042} C_VEL
LIN {X 0,Y 199.33,Z 345.033,A -85,B 0,C 180,E1 -23182.795,E2 -23182.795} C_VEL
LIN {X 0,Y 193.97,Z 335.364,A -85,B 0,C 180,E1 -23185.54,E2 -23185.54} C_VEL
LIN {X 0,Y 188.673,Z 327.75,A -85,B 0,C 180,E1 -23188.489,E2 -23188.489} C_VEL
LIN {X 0,Y 185.639,Z 323.6,A -85,B 0,C 180,E1 -23190.362,E2 -23190.362} C_VEL
LIN {X 0,Y 182.505,Z 319.433,A -85,B 0,C 180,E1 -23192.477,E2 -23192.477} C_VEL
LIN {X 0,Y 179.812,Z 316.172,A -85,B 0,C 180,E1 -23194.459,E2 -23194.459} C_VEL
LIN {X 0,Y 178.952,Z 314.761,A -85,B 0,C 180,E1 -23195.171,E2 -23195.171} C_VEL
LIN {X 0,Y 176.066,Z 312.011,A -85,B 0,C 180,E1 -23197.561,E2 -23197.561} C_VEL
LIN {X 0,Y 174.595,Z 309.384,A -85,B 0,C 180,E1 -23199.048,E2 -23199.048} C_VEL
LIN {X 0,Y 171.865,Z 307.269,A -85,B 0,C 180,E1 -23201.832,E2 -23201.832} C_VEL
LIN {X 0,Y 169.737,Z 303.734,A -85,B 0,C 180,E1 -23204.695,E2 -23204.695} C_VEL
LIN {X 0,Y 166.653,Z 301.55,A -85,B 0,C 180,E1 -23209.69,E2 -23209.69} C_VEL
LIN {X 0,Y 164.962,Z 298.355,A -85,B 0,C 180,E1 -23215.724,E2 -23215.724} C_VEL
LIN {X 0,Y 165.292,Z 297.64,A -85,B 0,C 180,E1 -23220,E2 -23220} C_VEL
LIN {X 0,Y 164.969,Z 298.106,A -85,B 0,C 180,E1 -23223.664,E2 -23223.664} C_VEL
LIN {X 0,Y 165.635,Z 300.152,A -85,B 0,C 180,E1 -23227.927,E2 -23227.927} C_VEL
LIN {X 0,Y 168.375,Z 303.074,A -85,B 0,C 180,E1 -23233.579,E2 -23233.579} C_VEL
LIN {X 0,Y 170.035,Z 304.063,A -85,B 0,C 180,E1 -23235.892,E2 -23235.892} C_VEL
LIN {X 0,Y 171.848,Z 307.24,A -85,B 0,C 180,E1 -23238.324,E2 -23238.324} C_VEL
LIN {X 0,Y 174.824,Z 309.766,A -85,B 0,C 180,E1 -23241.366,E2 -23241.366} C_VEL
LIN {X 0,Y 176.641,Z 312.739,A -85,B 0,C 180,E1 -23243.135,E2 -23243.135} C_VEL
LIN {X 0,Y 179.325,Z 315.308,A -85,B 0,C 180,E1 -23245.312,E2 -23245.312} C_VEL
LIN {X 0,Y 181.852,Z 318.825,A -85,B 0,C 180,E1 -23247.252,E2 -23247.252} C_VEL
LIN {X 0,Y 183.352,Z 320.489,A -85,B 0,C 180,E1 -23248.287,E2 -23248.287} C_VEL
LIN {X 0,Y 186.206,Z 324.172,A -85,B 0,C 180,E1 -23250.163,E2 -23250.163} C_VEL
LIN {X 0,Y 192.671,Z 333.33,A -85,B 0,C 180,E1 -23253.938,E2 -23253.938} C_VEL
LIN {X 0,Y 199.237,Z 343.516,A -85,B 0,C 180,E1 -23257.258,E2 -23257.258} C_VEL
LIN {X 0,Y 202.535,Z 349.597,A -85,B 0,C 180,E1 -23258.81,E2 -23258.81} C_VEL
LIN {X 0,Y 207.928,Z 361.266,A -85,B 0,C 180,E1 -23261.232,E2 -23261.232} C_VEL
LIN {X 0,Y 210.486,Z 367.706,A -85,B 0,C 180,E1 -23262.344,E2 -23262.344} C_VEL
LIN {X 0,Y 206.411,Z 427.338,A -85,B 0,C 180,E1 -23264.169,E2 -23264.169} C_VEL
LIN {X 0,Y 204.505,Z 441.237,A -85,B 0,C 180,E1 -23264.864,E2 -23264.864} C_VEL
LIN {X 0,Y 201.881,Z 454.757,A -85,B 0,C 180,E1 -23265.874,E2 -23265.874} C_VEL
LIN {X 0,Y 198.834,Z 467.052,A -85,B 0,C 180,E1 -23267.125,E2 -23267.125} C_VEL
LIN {X 0,Y 194.94,Z 479.933,A -85,B 0,C 180,E1 -23268.857,E2 -23268.857} C_VEL
LIN {X 0,Y 191.017,Z 491.277,A -85,B 0,C 180,E1 -23270.847,E2 -23270.847} C_VEL
LIN {X 0,Y 186.917,Z 501.335,A -85,B 0,C 180,E1 -23273.017,E2 -23273.017} C_VEL
LIN {X 0,Y 181.916,Z 512.085,A -85,B 0,C 180,E1 -23275.932,E2 -23275.932} C_VEL
LIN {X 0,Y 177.559,Z 520.955,A -85,B 0,C 180,E1 -23279.033,E2 -23279.033} C_VEL
LIN {X 0,Y 172.966,Z 529.449,A -85,B 0,C 180,E1 -23282.8,E2 -23282.8} C_VEL
LIN {X 0,Y 169.389,Z 536.287,A -85,B 0,C 180,E1 -23286.787,E2 -23286.787} C_VEL
LIN {X 0,Y 166.79,Z 541.005,A -85,B 0,C 180,E1 -23290.3,E2 -23290.3} C_VEL
LIN {X 0,Y 164.202,Z 545.892,A -85,B 0,C 180,E1 -23295.12,E2 -23295.12} C_VEL
LIN {X 0,Y 162.618,Z 549.29,A -85,B 0,C 180,E1 -23300.045,E2 -23300.045} C_VEL
LIN {X 0,Y 161.871,Z 551.303,A -85,B 0,C 180,E1 -23305.018,E2 -23305.018} C_VEL
LIN {X 0,Y 161.781,Z 551.986,A -85,B 0,C 180,E1 -23310,E2 -23310} C_VEL
LIN {X 0,Y 161.87,Z 551.352,A -85,B 0,C 180,E1 -23314.981,E2 -23314.981} C_VEL
LIN {X 0,Y 162.61,Z 549.383,A -85,B 0,C 180,E1 -23319.955,E2 -23319.955} C_VEL
LIN {X 0,Y 164.176,Z 546.031,A -85,B 0,C 180,E1 -23324.882,E2 -23324.882} C_VEL
LIN {X 0,Y 166.749,Z 541.196,A -85,B 0,C 180,E1 -23329.704,E2 -23329.704} C_VEL
LIN {X 0,Y 170.281,Z 534.724,A -85,B 0,C 180,E1 -23334.376,E2 -23334.376} C_VEL
LIN {X 0,Y 174.14,Z 527.517,A -85,B 0,C 180,E1 -23338.307,E2 -23338.307} C_VEL
LIN {X 0,Y 178.862,Z 518.597,A -85,B 0,C 180,E1 -23342.035,E2 -23342.035} C_VEL
LIN {X 0,Y 183.408,Z 509.224,A -85,B 0,C 180,E1 -23345.083,E2 -23345.083} C_VEL
LIN {X 0,Y 188.113,Z 498.844,A -85,B 0,C 180,E1 -23347.717,E2 -23347.717} C_VEL
LIN {X 0,Y 192.716,Z 486.888,A -85,B 0,C 180,E1 -23350.128,E2 -23350.128} C_VEL
LIN {X 0,Y 196.773,Z 474.685,A -85,B 0,C 180,E1 -23352.041,E2 -23352.041} C_VEL
LIN {X 0,Y 200.264,Z 462.316,A -85,B 0,C 180,E1 -23353.527,E2 -23353.527} C_VEL
LIN {X 0,Y 203.358,Z 448.587,A -85,B 0,C 180,E1 -23354.76,E2 -23354.76} C_VEL
LIN {X 0,Y 205.722,Z 434.244,A -85,B 0,C 180,E1 -23355.665,E2 -23355.665} C_VEL
LIN {X 0,Y 207.156,Z 420.171,A -85,B 0,C 180,E1 -23356.227,E2 -23356.227} C_VEL
LIN {X 0,Y 210.691,Z 367.912,A -85,B 0,C 180,E1 -23357.769,E2 -23357.769} C_VEL
LIN {X 0,Y 206.155,Z 357.056,A -85,B 0,C 180,E1 -23359.749,E2 -23359.749} C_VEL
LIN {X 0,Y 200.636,Z 345.736,A -85,B 0,C 180,E1 -23362.296,E2 -23362.296} C_VEL
LIN {X 0,Y 194.544,Z 336.067,A -85,B 0,C 180,E1 -23365.296,E2 -23365.296} C_VEL
LIN {X 0,Y 188.75,Z 327.769,A -85,B 0,C 180,E1 -23368.516,E2 -23368.516} C_VEL
LIN {X 0,Y 185.743,Z 323.692,A -85,B 0,C 180,E1 -23370.38,E2 -23370.38} C_VEL
LIN {X 0,Y 182.626,Z 319.533,A -85,B 0,C 180,E1 -23372.497,E2 -23372.497} C_VEL
LIN {X 0,Y 179.783,Z 316.094,A -85,B 0,C 180,E1 -23374.607,E2 -23374.607} C_VEL
LIN {X 0,Y 178.849,Z 314.692,A -85,B 0,C 180,E1 -23375.379,E2 -23375.379} C_VEL
LIN {X 0,Y 176.079,Z 311.956,A -85,B 0,C 180,E1 -23377.717,E2 -23377.717} C_VEL
LIN {X 0,Y 174.63,Z 309.396,A -85,B 0,C 180,E1 -23379.199,E2 -23379.199} C_VEL
LIN {X 0,Y 171.928,Z 307.344,A -85,B 0,C 180,E1 -23381.993,E2 -23381.993} C_VEL
LIN {X 0,Y 170.183,Z 304.377,A -85,B 0,C 180,E1 -23384.352,E2 -23384.352} C_VEL
LIN {X 0,Y 169.321,Z 303.504,A -85,B 0,C 180,E1 -23385.579,E2 -23385.579} C_VEL
LIN {X 0,Y 166.628,Z 301.526,A -85,B 0,C 180,E1 -23390.287,E2 -23390.287} C_VEL
LIN {X 0,Y 165.115,Z 298.16,A -85,B 0,C 180,E1 -23397.484,E2 -23397.484} C_VEL
LIN {X 0,Y 165.327,Z 297.795,A -85,B 0,C 180,E1 -23400,E2 -23400} C_VEL
LIN {X 0,Y 165.085,Z 298.363,A -85,B 0,C 180,E1 -23403.05,E2 -23403.05} C_VEL
LIN {X 0,Y 168.974,Z 303.327,A -85,B 0,C 180,E1 -23413.837,E2 -23413.837} C_VEL
LIN {X 0,Y 170.15,Z 304.223,A -85,B 0,C 180,E1 -23415.497,E2 -23415.497} C_VEL
LIN {X 0,Y 171.645,Z 306.965,A -85,B 0,C 180,E1 -23417.576,E2 -23417.576} C_VEL
LIN {X 0,Y 174.305,Z 309.24,A -85,B 0,C 180,E1 -23420.413,E2 -23420.413} C_VEL
LIN {X 0,Y 174.891,Z 309.827,A -85,B 0,C 180,E1 -23420.987,E2 -23420.987} C_VEL
LIN {X 0,Y 176.746,Z 312.851,A -85,B 0,C 180,E1 -23422.811,E2 -23422.811} C_VEL
LIN {X 0,Y 179.277,Z 315.213,A -85,B 0,C 180,E1 -23424.881,E2 -23424.881} C_VEL
LIN {X 0,Y 182,Z 318.922,A -85,B 0,C 180,E1 -23426.983,E2 -23426.983} C_VEL
LIN {X 0,Y 183.446,Z 320.603,A -85,B 0,C 180,E1 -23427.993,E2 -23427.993} C_VEL
LIN {X 0,Y 187.001,Z 325.395,A -85,B 0,C 180,E1 -23430.332,E2 -23430.332} C_VEL
LIN {X 0,Y 190.834,Z 330.792,A -85,B 0,C 180,E1 -23432.612,E2 -23432.612} C_VEL
LIN {X 0,Y 194.515,Z 336.097,A -85,B 0,C 180,E1 -23434.606,E2 -23434.606} C_VEL
LIN {X 0,Y 200.538,Z 347.186,A -85,B 0,C 180,E1 -23437.664,E2 -23437.664} C_VEL
LIN {X 0,Y 205.941,Z 358.699,A -85,B 0,C 180,E1 -23440.18,E2 -23440.18} C_VEL
LIN {X 0,Y 210.49,Z 370.059,A -85,B 0,C 180,E1 -23442.191,E2 -23442.191} C_VEL
LIN {X 0,Y 206.486,Z 429.607,A -85,B 0,C 180,E1 -23444.022,E2 -23444.022} C_VEL
LIN {X 0,Y 204.446,Z 444.382,A -85,B 0,C 180,E1 -23444.761,E2 -23444.761} C_VEL
LIN {X 0,Y 201.863,Z 457.237,A -85,B 0,C 180,E1 -23445.695,E2 -23445.695} C_VEL
LIN {X 0,Y 199.613,Z 466.423,A -85,B 0,C 180,E1 -23446.583,E2 -23446.583} C_VEL
LIN {X 0,Y 197.634,Z 471.777,A -85,B 0,C 180,E1 -23447.038,E2 -23447.038} C_VEL
LIN {X 0,Y 192.857,Z 480.295,A -85,B 0,C 180,E1 -23447.577,E2 -23447.577} C_VEL
LIN {X 0,Y 187.825,Z 488.458,A -85,B 0,C 180,E1 -23448.309,E2 -23448.309} C_VEL
LIN {X 0,Y 185.472,Z 493.25,A -85,B 0,C 180,E1 -23449.074,E2 -23449.074} C_VEL
LIN {X 0,Y 180.757,Z 504.448,A -85,B 0,C 180,E1 -23451.532,E2 -23451.532} C_VEL
LIN {X 0,Y 175.545,Z 515.16,A -85,B 0,C 180,E1 -23454.515,E2 -23454.515} C_VEL
LIN {X 0,Y 170.92,Z 524.004,A -85,B 0,C 180,E1 -23457.688,E2 -23457.688} C_VEL
LIN {X 0,Y 166.163,Z 532.482,A -85,B 0,C 180,E1 -23461.588,E2 -23461.588} C_VEL
LIN {X 0,Y 162.483,Z 538.993,A -85,B 0,C 180,E1 -23465.498,E2 -23465.498} C_VEL
LIN {X 0,Y 159.659,Z 544.021,A -85,B 0,C 180,E1 -23469.382,E2 -23469.382} C_VEL
LIN {X 0,Y 156.897,Z 548.899,A -85,B 0,C 180,E1 -23474.41,E2 -23474.41} C_VEL
LIN {X 0,Y 155.387,Z 552.292,A -85,B 0,C 180,E1 -23479.577,E2 -23479.577} C_VEL
LIN {X 0,Y 154.695,Z 554.296,A -85,B 0,C 180,E1 -23484.787,E2 -23484.787} C_VEL
LIN {X 0,Y 154.684,Z 554.955,A -85,B 0,C 180,E1 -23490,E2 -23490} C_VEL
LIN {X 0,Y 154.695,Z 554.274,A -85,B 0,C 180,E1 -23495.213,E2 -23495.213} C_VEL
LIN {X 0,Y 155.388,Z 552.25,A -85,B 0,C 180,E1 -23500.423,E2 -23500.423} C_VEL
LIN {X 0,Y 156.906,Z 548.834,A -85,B 0,C 180,E1 -23505.589,E2 -23505.589} C_VEL
LIN {X 0,Y 159.643,Z 543.927,A -85,B 0,C 180,E1 -23510.621,E2 -23510.621} C_VEL
LIN {X 0,Y 162.657,Z 538.363,A -85,B 0,C 180,E1 -23514.858,E2 -23514.858} C_VEL
LIN {X 0,Y 166.767,Z 531.219,A -85,B 0,C 180,E1 -23518.988,E2 -23518.988} C_VEL
LIN {X 0,Y 171.662,Z 522.471,A -85,B 0,C 180,E1 -23522.851,E2 -23522.851} C_VEL
LIN {X 0,Y 176.385,Z 513.317,A -85,B 0,C 180,E1 -23525.994,E2 -23525.994} C_VEL
LIN {X 0,Y 181.44,Z 502.787,A -85,B 0,C 180,E1 -23528.806,E2 -23528.806} C_VEL
LIN {X 0,Y 186.23,Z 490.864,A -85,B 0,C 180,E1 -23531.331,E2 -23531.331} C_VEL
LIN {X 0,Y 190.753,Z 478.318,A -85,B 0,C 180,E1 -23533.33,E2 -23533.33} C_VEL
LIN {X 0,Y 194.451,Z 466.169,A -85,B 0,C 180,E1 -23534.811,E2 -23534.811} C_VEL
LIN {X 0,Y 197.706,Z 452.789,A -85,B 0,C 180,E1 -23536.04,E2 -23536.04} C_VEL
LIN {X 0,Y 200.138,Z 439.081,A -85,B 0,C 180,E1 -23536.956,E2 -23536.956} C_VEL
LIN {X 0,Y 201.75,Z 426.113,A -85,B 0,C 180,E1 -23537.505,E2 -23537.505} C_VEL
LIN {X 0,Y 205.439,Z 373.476,A -85,B 0,C 180,E1 -23539.104,E2 -23539.104} C_VEL
LIN {X 0,Y 205.344,Z 371.868,A -85,B 0,C 180,E1 -23539.219,E2 -23539.219} C_VEL
LIN {X 0,Y 200.372,Z 359.643,A -85,B 0,C 180,E1 -23541.575,E2 -23541.575} C_VEL
LIN {X 0,Y 194.76,Z 347.947,A -85,B 0,C 180,E1 -23544.417,E2 -23544.417} C_VEL
LIN {X 0,Y 190.346,Z 339.999,A -85,B 0,C 180,E1 -23546.845,E2 -23546.845} C_VEL
LIN {X 0,Y 185.747,Z 333.266,A -85,B 0,C 180,E1 -23549.574,E2 -23549.574} C_VEL
LIN {X 0,Y 183.075,Z 329.497,A -85,B 0,C 180,E1 -23551.324,E2 -23551.324} C_VEL
LIN {X 0,Y 180.226,Z 325.602,A -85,B 0,C 180,E1 -23553.356,E2 -23553.356} C_VEL
LIN {X 0,Y 177.608,Z 322.222,A -85,B 0,C 180,E1 -23555.403,E2 -23555.403} C_VEL
LIN {X 0,Y 176.438,Z 320.837,A -85,B 0,C 180,E1 -23556.381,E2 -23556.381} C_VEL
LIN {X 0,Y 173.787,Z 317.725,A -85,B 0,C 180,E1 -23558.801,E2 -23558.801} C_VEL
LIN {X 0,Y 172.768,Z 316.005,A -85,B 0,C 180,E1 -23559.889,E2 -23559.889} C_VEL
LIN {X 0,Y 170.176,Z 313.666,A -85,B 0,C 180,E1 -23562.733,E2 -23562.733} C_VEL
LIN {X 0,Y 168.464,Z 310.603,A -85,B 0,C 180,E1 -23565.196,E2 -23565.196} C_VEL
LIN {X 0,Y 165.524,Z 308.398,A -85,B 0,C 180,E1 -23570.222,E2 -23570.222} C_VEL
LIN {X 0,Y 163.821,Z 305.222,A -85,B 0,C 180,E1 -23576.311,E2 -23576.311} C_VEL
LIN {X 0,Y 163.551,Z 304.529,A -85,B 0,C 180,E1 -23580,E2 -23580} C_VEL
LIN {X 0,Y 163.839,Z 305.28,A -85,B 0,C 180,E1 -23583.997,E2 -23583.997} C_VEL
LIN {X 0,Y 167.337,Z 310.066,A -85,B 0,C 180,E1 -23593.356,E2 -23593.356} C_VEL
LIN {X 0,Y 168.645,Z 310.855,A -85,B 0,C 180,E1 -23595.252,E2 -23595.252} C_VEL
LIN {X 0,Y 170.622,Z 314.247,A -85,B 0,C 180,E1 -23597.995,E2 -23597.995} C_VEL
LIN {X 0,Y 173.095,Z 316.419,A -85,B 0,C 180,E1 -23600.629,E2 -23600.629} C_VEL
LIN {X 0,Y 175.357,Z 319.811,A -85,B 0,C 180,E1 -23602.873,E2 -23602.873} C_VEL
LIN {X 0,Y 177.322,Z 321.738,A -85,B 0,C 180,E1 -23604.525,E2 -23604.525} C_VEL
LIN {X 0,Y 180.064,Z 325.498,A -85,B 0,C 180,E1 -23606.709,E2 -23606.709} C_VEL
LIN {X 0,Y 181.208,Z 326.901,A -85,B 0,C 180,E1 -23607.54,E2 -23607.54} C_VEL
LIN {X 0,Y 184.78,Z 331.852,A -85,B 0,C 180,E1 -23609.982,E2 -23609.982} C_VEL
LIN {X 0,Y 189.761,Z 339.001,A -85,B 0,C 180,E1 -23612.994,E2 -23612.994} C_VEL
LIN {X 0,Y 196.154,Z 349.222,A -85,B 0,C 180,E1 -23616.4,E2 -23616.4} C_VEL
LIN {X 0,Y 199.922,Z 356.65,A -85,B 0,C 180,E1 -23618.27,E2 -23618.27} C_VEL
LIN {X 0,Y 204.503,Z 367.175,A -85,B 0,C 180,E1 -23620.436,E2 -23620.436} C_VEL
LIN {X 0,Y 205.592,Z 369.909,A -85,B 0,C 180,E1 -23620.935,E2 -23620.935} C_VEL
LIN {X 0,Y 202.312,Z 418.107,A -85,B 0,C 180,E1 -23622.402,E2 -23622.402} C_VEL
LIN {X 0,Y 200.842,Z 433.27,A -85,B 0,C 180,E1 -23622.983,E2 -23622.983} C_VEL
LIN {X 0,Y 198.472,Z 447.294,A -85,B 0,C 180,E1 -23623.824,E2 -23623.824} C_VEL
LIN {X 0,Y 195.266,Z 461.346,A -85,B 0,C 180,E1 -23625.063,E2 -23625.063} C_VEL
LIN {X 0,Y 191.651,Z 473.933,A -85,B 0,C 180,E1 -23626.562,E2 -23626.562} C_VEL
LIN {X 0,Y 187.263,Z 486.738,A -85,B 0,C 180,E1 -23628.576,E2 -23628.576} C_VEL
LIN {X 0,Y 182.643,Z 498.351,A -85,B 0,C 180,E1 -23630.943,E2 -23630.943} C_VEL
LIN {X 0,Y 177.738,Z 508.826,A -85,B 0,C 180,E1 -23633.622,E2 -23633.622} C_VEL
LIN {X 0,Y 172.959,Z 518.278,A -85,B 0,C 180,E1 -23636.733,E2 -23636.733} C_VEL
LIN {X 0,Y 167.939,Z 527.292,A -85,B 0,C 180,E1 -23640.547,E2 -23640.547} C_VEL
LIN {X 0,Y 163.844,Z 534.552,A -85,B 0,C 180,E1 -23644.6,E2 -23644.6} C_VEL
LIN {X 0,Y 161.011,Z 539.634,A -85,B 0,C 180,E1 -23648.222,E2 -23648.222} C_VEL
LIN {X 0,Y 157.874,Z 544.899,A -85,B 0,C 180,E1 -23653.181,E2 -23653.181} C_VEL
LIN {X 0,Y 156.337,Z 547.837,A -85,B 0,C 180,E1 -23657.011,E2 -23657.011} C_VEL
LIN {X 0,Y 155.158,Z 550.531,A -85,B 0,C 180,E1 -23662.19,E2 -23662.19} C_VEL
LIN {X 0,Y 154.667,Z 551.876,A -85,B 0,C 180,E1 -23667.396,E2 -23667.396} C_VEL
LIN {X 0,Y 154.657,Z 551.986,A -85,B 0,C 180,E1 -23671.3,E2 -23671.3} C_VEL
LIN {X 0,Y 154.801,Z 551.419,A -85,B 0,C 180,E1 -23675.209,E2 -23675.209} C_VEL
LIN {X 0,Y 155.156,Z 550.602,A -85,B 0,C 180,E1 -23677.81,E2 -23677.81} C_VEL
LIN {X 0,Y 156.317,Z 547.95,A -85,B 0,C 180,E1 -23682.991,E2 -23682.991} C_VEL
LIN {X 0,Y 158.464,Z 543.874,A -85,B 0,C 180,E1 -23688.086,E2 -23688.086} C_VEL
LIN {X 0,Y 161.811,Z 538.242,A -85,B 0,C 180,E1 -23693.01,E2 -23693.01} C_VEL
LIN {X 0,Y 165.401,Z 531.911,A -85,B 0,C 180,E1 -23697.16,E2 -23697.16} C_VEL
LIN {X 0,Y 169.941,Z 523.975,A -85,B 0,C 180,E1 -23701.127,E2 -23701.127} C_VEL
LIN {X 0,Y 174.419,Z 515.7,A -85,B 0,C 180,E1 -23704.34,E2 -23704.34} C_VEL
LIN {X 0,Y 179.409,Z 505.73,A -85,B 0,C 180,E1 -23707.385,E2 -23707.385} C_VEL
LIN {X 0,Y 184.346,Z 494.627,A -85,B 0,C 180,E1 -23710.04,E2 -23710.04} C_VEL
LIN {X 0,Y 189.06,Z 482.162,A -85,B 0,C 180,E1 -23712.357,E2 -23712.357} C_VEL
LIN {X 0,Y 193.118,Z 469.8,A -85,B 0,C 180,E1 -23714.106,E2 -23714.106} C_VEL
LIN {X 0,Y 196.78,Z 456.005,A -85,B 0,C 180,E1 -23715.585,E2 -23715.585} C_VEL
LIN {X 0,Y 199.632,Z 442.13,A -85,B 0,C 180,E1 -23716.65,E2 -23716.65} C_VEL
LIN {X 0,Y 201.599,Z 427.964,A -85,B 0,C 180,E1 -23717.403,E2 -23717.403} C_VEL
LIN {X 0,Y 205.152,Z 380.247,A -85,B 0,C 180,E1 -23718.857,E2 -23718.857} C_VEL
LIN {X 0,Y 205.718,Z 370.065,A -85,B 0,C 180,E1 -23719.207,E2 -23719.207} C_VEL
LIN {X 0,Y 201.699,Z 360.364,A -85,B 0,C 180,E1 -23721.086,E2 -23721.086} C_VEL
LIN {X 0,Y 197.103,Z 350.745,A -85,B 0,C 180,E1 -23723.347,E2 -23723.347} C_VEL
LIN {X 0,Y 191.341,Z 341.385,A -85,B 0,C 180,E1 -23726.354,E2 -23726.354} C_VEL
LIN {X 0,Y 186.212,Z 333.792,A -85,B 0,C 180,E1 -23729.368,E2 -23729.368} C_VEL
LIN {X 0,Y 183.042,Z 329.416,A -85,B 0,C 180,E1 -23731.441,E2 -23731.441} C_VEL
LIN {X 0,Y 180.351,Z 325.74,A -85,B 0,C 180,E1 -23733.375,E2 -23733.375} C_VEL
LIN {X 0,Y 177.594,Z 322.166,A -85,B 0,C 180,E1 -23735.552,E2 -23735.552} C_VEL
LIN {X 0,Y 176.608,Z 320.961,A -85,B 0,C 180,E1 -23736.387,E2 -23736.387} C_VEL
LIN {X 0,Y 173.885,Z 317.824,A -85,B 0,C 180,E1 -23738.887,E2 -23738.887} C_VEL
LIN {X 0,Y 172.937,Z 316.103,A -85,B 0,C 180,E1 -23739.921,E2 -23739.921} C_VEL
LIN {X 0,Y 170.143,Z 313.595,A -85,B 0,C 180,E1 -23743.038,E2 -23743.038} C_VEL
LIN {X 0,Y 168.476,Z 310.613,A -85,B 0,C 180,E1 -23745.505,E2 -23745.505} C_VEL
LIN {X 0,Y 165.635,Z 308.529,A -85,B 0,C 180,E1 -23750.536,E2 -23750.536} C_VEL
LIN {X 0,Y 163.912,Z 305.025,A -85,B 0,C 180,E1 -23758.157,E2 -23758.157} C_VEL
LIN {X 0,Y 163.865,Z 304.753,A -85,B 0,C 180,E1 -23760,E2 -23760} C_VEL
LIN {X 0,Y 164.056,Z 305.576,A -85,B 0,C 180,E1 -23763.377,E2 -23763.377} C_VEL
LIN {X 0,Y 167.736,Z 310.233,A -85,B 0,C 180,E1 -23773.323,E2 -23773.323} C_VEL
LIN {X 0,Y 168.721,Z 310.943,A -85,B 0,C 180,E1 -23774.781,E2 -23774.781} C_VEL
LIN {X 0,Y 170.323,Z 313.769,A -85,B 0,C 180,E1 -23777.097,E2 -23777.097} C_VEL
LIN {X 0,Y 172.846,Z 316.032,A -85,B 0,C 180,E1 -23779.901,E2 -23779.901} C_VEL
LIN {X 0,Y 175.439,Z 319.896,A -85,B 0,C 180,E1 -23782.524,E2 -23782.524} C_VEL
LIN {X 0,Y 177.356,Z 321.771,A -85,B 0,C 180,E1 -23784.152,E2 -23784.152} C_VEL
LIN {X 0,Y 180.184,Z 325.569,A -85,B 0,C 180,E1 -23786.417,E2 -23786.417} C_VEL
LIN {X 0,Y 181.578,Z 327.39,A -85,B 0,C 180,E1 -23787.441,E2 -23787.441} C_VEL
LIN {X 0,Y 184.967,Z 332.101,A -85,B 0,C 180,E1 -23789.757,E2 -23789.757} C_VEL
LIN {X 0,Y 188.283,Z 336.895,A -85,B 0,C 180,E1 -23791.815,E2 -23791.815} C_VEL
LIN {X 0,Y 191.48,Z 341.684,A -85,B 0,C 180,E1 -23793.641,E2 -23793.641} C_VEL
LIN {X 0,Y 197.111,Z 352.37,A -85,B 0,C 180,E1 -23796.666,E2 -23796.666} C_VEL
LIN {X 0,Y 202.322,Z 363.932,A -85,B 0,C 180,E1 -23799.241,E2 -23799.241} C_VEL
LIN {X 0,Y 205.665,Z 372.453,A -85,B 0,C 180,E1 -23800.814,E2 -23800.814} C_VEL
LIN {X 0,Y 201.565,Z 430.07,A -85,B 0,C 180,E1 -23802.595,E2 -23802.595} C_VEL
LIN {X 0,Y 199.521,Z 444.325,A -85,B 0,C 180,E1 -23803.316,E2 -23803.316} C_VEL
LIN {X 0,Y 196.567,Z 458.307,A -85,B 0,C 180,E1 -23804.352,E2 -23804.352} C_VEL
LIN {X 0,Y 192.858,Z 472.179,A -85,B 0,C 180,E1 -23805.819,E2 -23805.819} C_VEL
LIN {X 0,Y 188.726,Z 484.6,A -85,B 0,C 180,E1 -23807.55,E2 -23807.55} C_VEL
LIN {X 0,Y 185.472,Z 493.25,A -85,B 0,C 180,E1 -23809.074,E2 -23809.074} C_VEL
LIN {X 0,Y 183.059,Z 498.006,A -85,B 0,C 180,E1 -23809.913,E2 -23809.913} C_VEL
LIN {X 0,Y 177.524,Z 505.427,A -85,B 0,C 180,E1 -23811.076,E2 -23811.076} C_VEL
LIN {X 0,Y 171.797,Z 512.425,A -85,B 0,C 180,E1 -23812.416,E2 -23812.416} C_VEL
LIN {X 0,Y 169.108,Z 516.387,A -85,B 0,C 180,E1 -23813.534,E2 -23813.534} C_VEL
LIN {X 0,Y 164.16,Z 525.295,A -85,B 0,C 180,E1 -23816.918,E2 -23816.918} C_VEL
LIN {X 0,Y 159.279,Z 533.497,A -85,B 0,C 180,E1 -23820.965,E2 -23820.965} C_VEL
LIN {X 0,Y 155.744,Z 539.373,A -85,B 0,C 180,E1 -23824.715,E2 -23824.715} C_VEL
LIN {X 0,Y 152.17,Z 545.344,A -85,B 0,C 180,E1 -23829.734,E2 -23829.734} C_VEL
LIN {X 0,Y 150.03,Z 548.833,A -85,B 0,C 180,E1 -23833.677,E2 -23833.677} C_VEL
LIN {X 0,Y 148.37,Z 552.226,A -85,B 0,C 180,E1 -23839.078,E2 -23839.078} C_VEL
LIN {X 0,Y 147.623,Z 554.23,A -85,B 0,C 180,E1 -23844.537,E2 -23844.537} C_VEL
LIN {X 0,Y 147.588,Z 554.888,A -85,B 0,C 180,E1 -23850,E2 -23850} C_VEL
LIN {X 0,Y 147.623,Z 554.207,A -85,B 0,C 180,E1 -23855.464,E2 -23855.464} C_VEL
LIN {X 0,Y 148.372,Z 552.182,A -85,B 0,C 180,E1 -23860.922,E2 -23860.922} C_VEL
LIN {X 0,Y 150.039,Z 548.766,A -85,B 0,C 180,E1 -23866.322,E2 -23866.322} C_VEL
LIN {X 0,Y 152.96,Z 543.859,A -85,B 0,C 180,E1 -23871.566,E2 -23871.566} C_VEL
LIN {X 0,Y 155.909,Z 538.768,A -85,B 0,C 180,E1 -23875.638,E2 -23875.638} C_VEL
LIN {X 0,Y 160.563,Z 531.15,A -85,B 0,C 180,E1 -23880.222,E2 -23880.222} C_VEL
LIN {X 0,Y 165.712,Z 522.402,A -85,B 0,C 180,E1 -23884.19,E2 -23884.19} C_VEL
LIN {X 0,Y 170.67,Z 513.247,A -85,B 0,C 180,E1 -23887.4,E2 -23887.4} C_VEL
LIN {X 0,Y 175.863,Z 502.89,A -85,B 0,C 180,E1 -23890.217,E2 -23890.217} C_VEL
LIN {X 0,Y 180.457,Z 492.051,A -85,B 0,C 180,E1 -23892.584,E2 -23892.584} C_VEL
LIN {X 0,Y 185.114,Z 479.829,A -85,B 0,C 180,E1 -23894.616,E2 -23894.616} C_VEL
LIN {X 0,Y 188.935,Z 468.077,A -85,B 0,C 180,E1 -23896.112,E2 -23896.112} C_VEL
LIN {X 0,Y 192.276,Z 455.313,A -85,B 0,C 180,E1 -23897.357,E2 -23897.357} C_VEL
LIN {X 0,Y 195.085,Z 440.833,A -85,B 0,C 180,E1 -23898.375,E2 -23898.375} C_VEL
LIN {X 0,Y 197.007,Z 426.253,A -85,B 0,C 180,E1 -23899.018,E2 -23899.018} C_VEL
LIN {X 0,Y 200.735,Z 374.62,A -85,B 0,C 180,E1 -23900.612,E2 -23900.612} C_VEL
LIN {X 0,Y 196.345,Z 363.603,A -85,B 0,C 180,E1 -23902.841,E2 -23902.841} C_VEL
LIN {X 0,Y 191.287,Z 352.766,A -85,B 0,C 180,E1 -23905.579,E2 -23905.579} C_VEL
LIN {X 0,Y 187.2,Z 345.191,A -85,B 0,C 180,E1 -23907.975,E2 -23907.975} C_VEL
LIN {X 0,Y 182.74,Z 338.564,A -85,B 0,C 180,E1 -23910.794,E2 -23910.794} C_VEL
LIN {X 0,Y 180.205,Z 334.947,A -85,B 0,C 180,E1 -23912.569,E2 -23912.569} C_VEL
LIN {X 0,Y 177.986,Z 331.811,A -85,B 0,C 180,E1 -23914.256,E2 -23914.256} C_VEL
LIN {X 0,Y 174.819,Z 327.55,A -85,B 0,C 180,E1 -23916.923,E2 -23916.923} C_VEL
LIN {X 0,Y 172.146,Z 324.37,A -85,B 0,C 180,E1 -23919.465,E2 -23919.465} C_VEL
LIN {X 0,Y 171.135,Z 322.704,A -85,B 0,C 180,E1 -23920.589,E2 -23920.589} C_VEL
LIN {X 0,Y 168.533,Z 320.044,A -85,B 0,C 180,E1 -23923.651,E2 -23923.651} C_VEL
LIN {X 0,Y 167.204,Z 317.465,A -85,B 0,C 180,E1 -23925.704,E2 -23925.704} C_VEL
LIN {X 0,Y 164.527,Z 315.405,A -85,B 0,C 180,E1 -23930.472,E2 -23930.472} C_VEL
LIN {X 0,Y 162.909,Z 312.215,A -85,B 0,C 180,E1 -23936.599,E2 -23936.599} C_VEL
LIN {X 0,Y 162.685,Z 311.581,A -85,B 0,C 180,E1 -23940,E2 -23940} C_VEL
LIN {X 0,Y 162.925,Z 312.275,A -85,B 0,C 180,E1 -23943.71,E2 -23943.71} C_VEL
LIN {X 0,Y 166.119,Z 316.942,A -85,B 0,C 180,E1 -23952.833,E2 -23952.833} C_VEL
LIN {X 0,Y 167.274,Z 317.674,A -85,B 0,C 180,E1 -23954.601,E2 -23954.601} C_VEL
LIN {X 0,Y 169.524,Z 321.345,A -85,B 0,C 180,E1 -23957.803,E2 -23957.803} C_VEL
LIN {X 0,Y 171.478,Z 323.157,A -85,B 0,C 180,E1 -23959.964,E2 -23959.964} C_VEL
LIN {X 0,Y 173.878,Z 326.659,A -85,B 0,C 180,E1 -23962.424,E2 -23962.424} C_VEL
LIN {X 0,Y 175.487,Z 328.407,A -85,B 0,C 180,E1 -23963.844,E2 -23963.844} C_VEL
LIN {X 0,Y 178.291,Z 332.152,A -85,B 0,C 180,E1 -23966.153,E2 -23966.153} C_VEL
LIN {X 0,Y 182.517,Z 338.164,A -85,B 0,C 180,E1 -23969.226,E2 -23969.226} C_VEL
LIN {X 0,Y 187.08,Z 344.968,A -85,B 0,C 180,E1 -23972.128,E2 -23972.128} C_VEL
LIN {X 0,Y 192.929,Z 354.585,A -85,B 0,C 180,E1 -23975.415,E2 -23975.415} C_VEL
LIN {X 0,Y 196.16,Z 361.163,A -85,B 0,C 180,E1 -23977.12,E2 -23977.12} C_VEL
LIN {X 0,Y 200.86,Z 372.427,A -85,B 0,C 180,E1 -23979.488,E2 -23979.488} C_VEL
LIN {X 0,Y 197.215,Z 422.754,A -85,B 0,C 180,E1 -23981.027,E2 -23981.027} C_VEL
LIN {X 0,Y 195.486,Z 437.06,A -85,B 0,C 180,E1 -23981.66,E2 -23981.66} C_VEL
LIN {X 0,Y 193.095,Z 449.968,A -85,B 0,C 180,E1 -23982.522,E2 -23982.522} C_VEL
LIN {X 0,Y 189.785,Z 463.405,A -85,B 0,C 180,E1 -23983.772,E2 -23983.772} C_VEL
LIN {X 0,Y 186.05,Z 475.585,A -85,B 0,C 180,E1 -23985.288,E2 -23985.288} C_VEL
LIN {X 0,Y 181.827,Z 487.226,A -85,B 0,C 180,E1 -23987.169,E2 -23987.169} C_VEL
LIN {X 0,Y 177.191,Z 498.421,A -85,B 0,C 180,E1 -23989.498,E2 -23989.498} C_VEL
LIN {X 0,Y 172.065,Z 508.895,A -85,B 0,C 180,E1 -23992.218,E2 -23992.218} C_VEL
LIN {X 0,Y 167.047,Z 518.348,A -85,B 0,C 180,E1 -23995.392,E2 -23995.392} C_VEL
LIN {X 0,Y 161.771,Z 527.36,A -85,B 0,C 180,E1 -23999.306,E2 -23999.306} C_VEL
LIN {X 0,Y 157.416,Z 534.621,A -85,B 0,C 180,E1 -24003.484,E2 -24003.484} C_VEL
LIN {X 0,Y 154.413,Z 539.702,A -85,B 0,C 180,E1 -24007.24,E2 -24007.24} C_VEL
LIN {X 0,Y 151.046,Z 544.967,A -85,B 0,C 180,E1 -24012.396,E2 -24012.396} C_VEL
LIN {X 0,Y 149.411,Z 547.904,A -85,B 0,C 180,E1 -24016.397,E2 -24016.397} C_VEL
LIN {X 0,Y 148.099,Z 550.599,A -85,B 0,C 180,E1 -24021.815,E2 -24021.815} C_VEL
LIN {X 0,Y 147.572,Z 551.943,A -85,B 0,C 180,E1 -24027.27,E2 -24027.27} C_VEL
LIN {X 0,Y 147.597,Z 552.096,A -85,B 0,C 180,E1 -24030.613,E2 -24030.613} C_VEL
LIN {X 0,Y 147.726,Z 551.485,A -85,B 0,C 180,E1 -24035.46,E2 -24035.46} C_VEL
LIN {X 0,Y 148.604,Z 549.515,A -85,B 0,C 180,E1 -24040.904,E2 -24040.904} C_VEL
LIN {X 0,Y 150.419,Z 546.163,A -85,B 0,C 180,E1 -24046.28,E2 -24046.28} C_VEL
LIN {X 0,Y 153.41,Z 541.327,A -85,B 0,C 180,E1 -24051.499,E2 -24051.499} C_VEL
LIN {X 0,Y 157.341,Z 534.856,A -85,B 0,C 180,E1 -24056.53,E2 -24056.53} C_VEL
LIN {X 0,Y 161.728,Z 527.647,A -85,B 0,C 180,E1 -24060.703,E2 -24060.703} C_VEL
LIN {X 0,Y 166.951,Z 518.726,A -85,B 0,C 180,E1 -24064.631,E2 -24064.631} C_VEL
LIN {X 0,Y 171.975,Z 509.352,A -85,B 0,C 180,E1 -24067.805,E2 -24067.805} C_VEL
LIN {X 0,Y 177.091,Z 498.97,A -85,B 0,C 180,E1 -24070.529,E2 -24070.529} C_VEL
LIN {X 0,Y 181.955,Z 487.322,A -85,B 0,C 180,E1 -24072.958,E2 -24072.958} C_VEL
LIN {X 0,Y 186.463,Z 474.808,A -85,B 0,C 180,E1 -24074.966,E2 -24074.966} C_VEL
LIN {X 0,Y 190.24,Z 462.436,A -85,B 0,C 180,E1 -24076.468,E2 -24076.468} C_VEL
LIN {X 0,Y 193.524,Z 448.703,A -85,B 0,C 180,E1 -24077.724,E2 -24077.724} C_VEL
LIN {X 0,Y 196.074,Z 434.353,A -85,B 0,C 180,E1 -24078.63,E2 -24078.63} C_VEL
LIN {X 0,Y 197.63,Z 420.117,A -85,B 0,C 180,E1 -24079.199,E2 -24079.199} C_VEL
LIN {X 0,Y 201.034,Z 373.816,A -85,B 0,C 180,E1 -24080.574,E2 -24080.574} C_VEL
LIN {X 0,Y 200.89,Z 372.294,A -85,B 0,C 180,E1 -24080.708,E2 -24080.708} C_VEL
LIN {X 0,Y 197.147,Z 363.146,A -85,B 0,C 180,E1 -24082.594,E2 -24082.594} C_VEL
LIN {X 0,Y 193.345,Z 355.16,A -85,B 0,C 180,E1 -24084.595,E2 -24084.595} C_VEL
LIN {X 0,Y 186.75,Z 344.328,A -85,B 0,C 180,E1 -24088.325,E2 -24088.325} C_VEL
LIN {X 0,Y 181.322,Z 336.267,A -85,B 0,C 180,E1 -24091.888,E2 -24091.888} C_VEL
LIN {X 0,Y 178.12,Z 331.933,A -85,B 0,C 180,E1 -24094.277,E2 -24094.277} C_VEL
LIN {X 0,Y 174.917,Z 327.609,A -85,B 0,C 180,E1 -24096.996,E2 -24096.996} C_VEL
LIN {X 0,Y 172.101,Z 324.227,A -85,B 0,C 180,E1 -24099.716,E2 -24099.716} C_VEL
LIN {X 0,Y 171.254,Z 322.764,A -85,B 0,C 180,E1 -24100.681,E2 -24100.681} C_VEL
LIN {X 0,Y 168.363,Z 319.784,A -85,B 0,C 180,E1 -24104.179,E2 -24104.179} C_VEL
LIN {X 0,Y 167.226,Z 317.491,A -85,B 0,C 180,E1 -24106.016,E2 -24106.016} C_VEL
LIN {X 0,Y 164.526,Z 315.371,A -85,B 0,C 180,E1 -24111.092,E2 -24111.092} C_VEL
LIN {X 0,Y 163.044,Z 312.101,A -85,B 0,C 180,E1 -24118.147,E2 -24118.147} C_VEL
LIN {X 0,Y 162.998,Z 311.809,A -85,B 0,C 180,E1 -24120,E2 -24120} C_VEL
LIN {X 0,Y 163.182,Z 312.706,A -85,B 0,C 180,E1 -24123.395,E2 -24123.395} C_VEL
LIN {X 0,Y 166.698,Z 317.227,A -85,B 0,C 180,E1 -24133.097,E2 -24133.097} C_VEL
LIN {X 0,Y 167.406,Z 317.831,A -85,B 0,C 180,E1 -24134.201,E2 -24134.201} C_VEL
LIN {X 0,Y 169.45,Z 321.204,A -85,B 0,C 180,E1 -24137.188,E2 -24137.188} C_VEL
LIN {X 0,Y 171.572,Z 323.228,A -85,B 0,C 180,E1 -24139.591,E2 -24139.591} C_VEL
LIN {X 0,Y 173.844,Z 326.597,A -85,B 0,C 180,E1 -24141.959,E2 -24141.959} C_VEL
LIN {X 0,Y 175.588,Z 328.471,A -85,B 0,C 180,E1 -24143.516,E2 -24143.516} C_VEL
LIN {X 0,Y 179.395,Z 333.647,A -85,B 0,C 180,E1 -24146.62,E2 -24146.62} C_VEL
LIN {X 0,Y 182.731,Z 338.432,A -85,B 0,C 180,E1 -24149.015,E2 -24149.015} C_VEL
LIN {X 0,Y 187.495,Z 345.567,A -85,B 0,C 180,E1 -24152.043,E2 -24152.043} C_VEL
LIN {X 0,Y 192.384,Z 354.731,A -85,B 0,C 180,E1 -24154.885,E2 -24154.885} C_VEL
LIN {X 0,Y 196.89,Z 364.651,A -85,B 0,C 180,E1 -24157.31,E2 -24157.31} C_VEL
LIN {X 0,Y 200.906,Z 374.738,A -85,B 0,C 180,E1 -24159.345,E2 -24159.345} C_VEL
LIN {X 0,Y 196.853,Z 429.799,A -85,B 0,C 180,E1 -24161.063,E2 -24161.063} C_VEL
LIN {X 0,Y 194.71,Z 444.268,A -85,B 0,C 180,E1 -24161.792,E2 -24161.792} C_VEL
LIN {X 0,Y 191.668,Z 458.247,A -85,B 0,C 180,E1 -24162.834,E2 -24162.834} C_VEL
LIN {X 0,Y 187.82,Z 472.117,A -85,B 0,C 180,E1 -24164.306,E2 -24164.306} C_VEL
LIN {X 0,Y 183.537,Z 484.538,A -85,B 0,C 180,E1 -24166.051,E2 -24166.051} C_VEL
LIN {X 0,Y 179.017,Z 495.896,A -85,B 0,C 180,E1 -24168.135,E2 -24168.135} C_VEL
LIN {X 0,Y 174.313,Z 506.336,A -85,B 0,C 180,E1 -24170.58,E2 -24170.58} C_VEL
LIN {X 0,Y 169.108,Z 516.387,A -85,B 0,C 180,E1 -24173.534,E2 -24173.534} C_VEL
LIN {X 0,Y 166.417,Z 520.291,A -85,B 0,C 180,E1 -24174.743,E2 -24174.743} C_VEL
LIN {X 0,Y 160.567,Z 526.25,A -85,B 0,C 180,E1 -24176.623,E2 -24176.623} C_VEL
LIN {X 0,Y 154.785,Z 531.658,A -85,B 0,C 180,E1 -24178.79,E2 -24178.79} C_VEL
LIN {X 0,Y 152.27,Z 534.677,A -85,B 0,C 180,E1 -24180.432,E2 -24180.432} C_VEL
LIN {X 0,Y 148.361,Z 540.846,A -85,B 0,C 180,E1 -24184.765,E2 -24184.765} C_VEL
LIN {X 0,Y 144.654,Z 546.522,A -85,B 0,C 180,E1 -24190.118,E2 -24190.118} C_VEL
LIN {X 0,Y 142.148,Z 550.641,A -85,B 0,C 180,E1 -24195.688,E2 -24195.688} C_VEL
LIN {X 0,Y 140.844,Z 553.331,A -85,B 0,C 180,E1 -24201.391,E2 -24201.391} C_VEL
LIN {X 0,Y 140.42,Z 554.659,A -85,B 0,C 180,E1 -24207.131,E2 -24207.131} C_VEL
LIN {X 0,Y 140.484,Z 554.821,A -85,B 0,C 180,E1 -24210,E2 -24210} C_VEL
LIN {X 0,Y 140.547,Z 554.14,A -85,B 0,C 180,E1 -24215.74,E2 -24215.74} C_VEL
LIN {X 0,Y 141.379,Z 552.115,A -85,B 0,C 180,E1 -24221.469,E2 -24221.469} C_VEL
LIN {X 0,Y 143.198,Z 548.699,A -85,B 0,C 180,E1 -24227.126,E2 -24227.126} C_VEL
LIN {X 0,Y 146.326,Z 543.791,A -85,B 0,C 180,E1 -24232.596,E2 -24232.596} C_VEL
LIN {X 0,Y 150.505,Z 537.245,A -85,B 0,C 180,E1 -24237.837,E2 -24237.837} C_VEL
LIN {X 0,Y 155.183,Z 529.964,A -85,B 0,C 180,E1 -24242.149,E2 -24242.149} C_VEL
LIN {X 0,Y 160.645,Z 520.941,A -85,B 0,C 180,E1 -24246.199,E2 -24246.199} C_VEL
LIN {X 0,Y 166.019,Z 511.478,A -85,B 0,C 180,E1 -24249.418,E2 -24249.418} C_VEL
LIN {X 0,Y 171.612,Z 500.303,A -85,B 0,C 180,E1 -24252.37,E2 -24252.37} C_VEL
LIN {X 0,Y 176.854,Z 488.139,A -85,B 0,C 180,E1 -24254.858,E2 -24254.858} C_VEL
LIN {X 0,Y 181.245,Z 476.592,A -85,B 0,C 180,E1 -24256.639,E2 -24256.639} C_VEL
LIN {X 0,Y 185.492,Z 463.039,A -85,B 0,C 180,E1 -24258.238,E2 -24258.238} C_VEL
LIN {X 0,Y 188.71,Z 450.038,A -85,B 0,C 180,E1 -24259.358,E2 -24259.358} C_VEL
LIN {X 0,Y 191.226,Z 436.173,A -85,B 0,C 180,E1 -24260.205,E2 -24260.205} C_VEL
LIN {X 0,Y 192.788,Z 422.239,A -85,B 0,C 180,E1 -24260.746,E2 -24260.746} C_VEL
LIN {X 0,Y 196.091,Z 377.882,A -85,B 0,C 180,E1 -24262.099,E2 -24262.099} C_VEL
LIN {X 0,Y 195.864,Z 376.391,A -85,B 0,C 180,E1 -24262.271,E2 -24262.271} C_VEL
LIN {X 0,Y 191.998,Z 366.627,A -85,B 0,C 180,E1 -24264.392,E2 -24264.392} C_VEL
LIN {X 0,Y 187.628,Z 357.067,A -85,B 0,C 180,E1 -24266.943,E2 -24266.943} C_VEL
LIN {X 0,Y 184.131,Z 350.426,A -85,B 0,C 180,E1 -24269.139,E2 -24269.139} C_VEL
LIN {X 0,Y 178.813,Z 342.212,A -85,B 0,C 180,E1 -24272.807,E2 -24272.807} C_VEL
LIN {X 0,Y 175.794,Z 337.995,A -85,B 0,C 180,E1 -24275.18,E2 -24275.18} C_VEL
LIN {X 0,Y 172.863,Z 333.945,A -85,B 0,C 180,E1 -24277.792,E2 -24277.792} C_VEL
LIN {X 0,Y 170.171,Z 330.411,A -85,B 0,C 180,E1 -24280.55,E2 -24280.55} C_VEL
LIN {X 0,Y 169.437,Z 329.297,A -85,B 0,C 180,E1 -24281.406,E2 -24281.406} C_VEL
LIN {X 0,Y 166.928,Z 326.406,A -85,B 0,C 180,E1 -24284.598,E2 -24284.598} C_VEL
LIN {X 0,Y 165.754,Z 324.293,A -85,B 0,C 180,E1 -24286.515,E2 -24286.515} C_VEL
LIN {X 0,Y 163.031,Z 321.64,A -85,B 0,C 180,E1 -24292.102,E2 -24292.102} C_VEL
LIN {X 0,Y 161.983,Z 319.156,A -85,B 0,C 180,E1 -24297.047,E2 -24297.047} C_VEL
LIN {X 0,Y 161.819,Z 318.634,A -85,B 0,C 180,E1 -24300,E2 -24300} C_VEL
LIN {X 0,Y 162.072,Z 319.422,A -85,B 0,C 180,E1 -24303.854,E2 -24303.854} C_VEL
LIN {X 0,Y 165.09,Z 323.934,A -85,B 0,C 180,E1 -24312.602,E2 -24312.602} C_VEL
LIN {X 0,Y 165.996,Z 324.574,A -85,B 0,C 180,E1 -24314.055,E2 -24314.055} C_VEL
LIN {X 0,Y 168.197,Z 328.173,A -85,B 0,C 180,E1 -24317.321,E2 -24317.321} C_VEL
LIN {X 0,Y 169.858,Z 329.813,A -85,B 0,C 180,E1 -24319.252,E2 -24319.252} C_VEL
LIN {X 0,Y 172.439,Z 333.506,A -85,B 0,C 180,E1 -24321.991,E2 -24321.991} C_VEL
LIN {X 0,Y 173.764,Z 335.169,A -85,B 0,C 180,E1 -24323.225,E2 -24323.225} C_VEL
LIN {X 0,Y 177.037,Z 339.721,A -85,B 0,C 180,E1 -24326.007,E2 -24326.007} C_VEL
LIN {X 0,Y 180.643,Z 344.99,A -85,B 0,C 180,E1 -24328.701,E2 -24328.701} C_VEL
LIN {X 0,Y 185.875,Z 353.195,A -85,B 0,C 180,E1 -24332.121,E2 -24332.121} C_VEL
LIN {X 0,Y 190.987,Z 362.322,A -85,B 0,C 180,E1 -24335.085,E2 -24335.085} C_VEL
LIN {X 0,Y 195.88,Z 373.865,A -85,B 0,C 180,E1 -24337.764,E2 -24337.764} C_VEL
LIN {X 0,Y 196.216,Z 374.827,A -85,B 0,C 180,E1 -24337.947,E2 -24337.947} C_VEL
LIN {X 0,Y 193.122,Z 417.331,A -85,B 0,C 180,E1 -24339.269,E2 -24339.269} C_VEL
LIN {X 0,Y 191.61,Z 432.305,A -85,B 0,C 180,E1 -24339.83,E2 -24339.83} C_VEL
LIN {X 0,Y 189.219,Z 446.033,A -85,B 0,C 180,E1 -24340.617,E2 -24340.617} C_VEL
LIN {X 0,Y 186.064,Z 459.482,A -85,B 0,C 180,E1 -24341.757,E2 -24341.757} C_VEL
LIN {X 0,Y 182.144,Z 472.497,A -85,B 0,C 180,E1 -24343.258,E2 -24343.258} C_VEL
LIN {X 0,Y 177.452,Z 485.358,A -85,B 0,C 180,E1 -24345.248,E2 -24345.248} C_VEL
LIN {X 0,Y 172.349,Z 497.423,A -85,B 0,C 180,E1 -24347.715,E2 -24347.715} C_VEL
LIN {X 0,Y 167.469,Z 507.186,A -85,B 0,C 180,E1 -24350.211,E2 -24350.211} C_VEL
LIN {X 0,Y 162.088,Z 516.934,A -85,B 0,C 180,E1 -24353.403,E2 -24353.403} C_VEL
LIN {X 0,Y 157.216,Z 525.02,A -85,B 0,C 180,E1 -24356.798,E2 -24356.798} C_VEL
LIN {X 0,Y 152.114,Z 532.963,A -85,B 0,C 180,E1 -24361.131,E2 -24361.131} C_VEL
LIN {X 0,Y 147.862,Z 539.771,A -85,B 0,C 180,E1 -24366.171,E2 -24366.171} C_VEL
LIN {X 0,Y 144.262,Z 545.035,A -85,B 0,C 180,E1 -24371.539,E2 -24371.539} C_VEL
LIN {X 0,Y 142.494,Z 547.972,A -85,B 0,C 180,E1 -24375.723,E2 -24375.723} C_VEL
LIN {X 0,Y 141.058,Z 550.666,A -85,B 0,C 180,E1 -24381.404,E2 -24381.404} C_VEL
LIN {X 0,Y 140.491,Z 552.01,A -85,B 0,C 180,E1 -24387.132,E2 -24387.132} C_VEL
LIN {X 0,Y 140.524,Z 552.186,A -85,B 0,C 180,E1 -24390,E2 -24390} C_VEL
LIN {X 0,Y 140.654,Z 551.551,A -85,B 0,C 180,E1 -24395.735,E2 -24395.735} C_VEL
LIN {X 0,Y 141.625,Z 549.581,A -85,B 0,C 180,E1 -24401.449,E2 -24401.449} C_VEL
LIN {X 0,Y 143.572,Z 546.229,A -85,B 0,C 180,E1 -24407.079,E2 -24407.079} C_VEL
LIN {X 0,Y 146.808,Z 541.393,A -85,B 0,C 180,E1 -24412.517,E2 -24412.517} C_VEL
LIN {X 0,Y 150.976,Z 534.921,A -85,B 0,C 180,E1 -24417.742,E2 -24417.742} C_VEL
LIN {X 0,Y 155.639,Z 527.712,A -85,B 0,C 180,E1 -24422.044,E2 -24422.044} C_VEL
LIN {X 0,Y 161.149,Z 518.791,A -85,B 0,C 180,E1 -24426.068,E2 -24426.068} C_VEL
LIN {X 0,Y 166.427,Z 509.415,A -85,B 0,C 180,E1 -24429.303,E2 -24429.303} C_VEL
LIN {X 0,Y 171.752,Z 499.033,A -85,B 0,C 180,E1 -24432.07,E2 -24432.07} C_VEL
LIN {X 0,Y 176.579,Z 487.963,A -85,B 0,C 180,E1 -24434.426,E2 -24434.426} C_VEL
LIN {X 0,Y 180.974,Z 476.449,A -85,B 0,C 180,E1 -24436.325,E2 -24436.325} C_VEL
LIN {X 0,Y 184.868,Z 464.481,A -85,B 0,C 180,E1 -24437.842,E2 -24437.842} C_VEL
LIN {X 0,Y 188.255,Z 451.361,A -85,B 0,C 180,E1 -24439.109,E2 -24439.109} C_VEL
LIN {X 0,Y 191.058,Z 437.153,A -85,B 0,C 180,E1 -24440.059,E2 -24440.059} C_VEL
LIN {X 0,Y 192.807,Z 422.647,A -85,B 0,C 180,E1 -24440.721,E2 -24440.721} C_VEL
LIN {X 0,Y 196.442,Z 375.932,A -85,B 0,C 180,E1 -24442.112,E2 -24442.112} C_VEL
LIN {X 0,Y 196.197,Z 374.487,A -85,B 0,C 180,E1 -24442.289,E2 -24442.289} C_VEL
LIN {X 0,Y 191.833,Z 364.007,A -85,B 0,C 180,E1 -24444.671,E2 -24444.671} C_VEL
LIN {X 0,Y 189.034,Z 358.522,A -85,B 0,C 180,E1 -24446.254,E2 -24446.254} C_VEL
LIN {X 0,Y 183.748,Z 349.707,A -85,B 0,C 180,E1 -24449.47,E2 -24449.47} C_VEL
LIN {X 0,Y 178.935,Z 342.29,A -85,B 0,C 180,E1 -24452.832,E2 -24452.832} C_VEL
LIN {X 0,Y 175.937,Z 338.109,A -85,B 0,C 180,E1 -24455.201,E2 -24455.201} C_VEL
LIN {X 0,Y 172.89,Z 333.904,A -85,B 0,C 180,E1 -24457.943,E2 -24457.943} C_VEL
LIN {X 0,Y 170.287,Z 330.505,A -85,B 0,C 180,E1 -24460.642,E2 -24460.642} C_VEL
LIN {X 0,Y 169.503,Z 329.314,A -85,B 0,C 180,E1 -24461.569,E2 -24461.569} C_VEL
LIN {X 0,Y 166.843,Z 326.235,A -85,B 0,C 180,E1 -24465.048,E2 -24465.048} C_VEL
LIN {X 0,Y 165.798,Z 324.295,A -85,B 0,C 180,E1 -24466.83,E2 -24466.83} C_VEL
LIN {X 0,Y 162.99,Z 321.556,A -85,B 0,C 180,E1 -24473.034,E2 -24473.034} C_VEL
LIN {X 0,Y 162.145,Z 319.047,A -85,B 0,C 180,E1 -24478.758,E2 -24478.758} C_VEL
LIN {X 0,Y 162.151,Z 319.038,A -85,B 0,C 180,E1 -24481.242,E2 -24481.242} C_VEL
LIN {X 0,Y 166.113,Z 324.682,A -85,B 0,C 180,E1 -24493.612,E2 -24493.612} C_VEL
LIN {X 0,Y 168.248,Z 328.151,A -85,B 0,C 180,E1 -24496.845,E2 -24496.845} C_VEL
LIN {X 0,Y 169.999,Z 329.951,A -85,B 0,C 180,E1 -24498.921,E2 -24498.921} C_VEL
LIN {X 0,Y 172.411,Z 333.449,A -85,B 0,C 180,E1 -24501.522,E2 -24501.522} C_VEL
LIN {X 0,Y 173.838,Z 335.148,A -85,B 0,C 180,E1 -24502.86,E2 -24502.86} C_VEL
LIN {X 0,Y 177.165,Z 339.798,A -85,B 0,C 180,E1 -24505.714,E2 -24505.714} C_VEL
LIN {X 0,Y 181.741,Z 346.5,A -85,B 0,C 180,E1 -24509.096,E2 -24509.096} C_VEL
LIN {X 0,Y 185.778,Z 353.185,A -85,B 0,C 180,E1 -24511.741,E2 -24511.741} C_VEL
LIN {X 0,Y 190.344,Z 362.539,A -85,B 0,C 180,E1 -24514.509,E2 -24514.509} C_VEL
LIN {X 0,Y 194.575,Z 372.606,A -85,B 0,C 180,E1 -24516.888,E2 -24516.888} C_VEL
LIN {X 0,Y 196.289,Z 377.135,A -85,B 0,C 180,E1 -24517.814,E2 -24517.814} C_VEL
LIN {X 0,Y 192.262,Z 429.726,A -85,B 0,C 180,E1 -24519.465,E2 -24519.465} C_VEL
LIN {X 0,Y 190.044,Z 444.211,A -85,B 0,C 180,E1 -24520.194,E2 -24520.194} C_VEL
LIN {X 0,Y 186.915,Z 458.188,A -85,B 0,C 180,E1 -24521.238,E2 -24521.238} C_VEL
LIN {X 0,Y 182.928,Z 472.056,A -85,B 0,C 180,E1 -24522.714,E2 -24522.714} C_VEL
LIN {X 0,Y 178.489,Z 484.476,A -85,B 0,C 180,E1 -24524.467,E2 -24524.467} C_VEL
LIN {X 0,Y 173.788,Z 495.833,A -85,B 0,C 180,E1 -24526.57,E2 -24526.57} C_VEL
LIN {X 0,Y 168.861,Z 506.272,A -85,B 0,C 180,E1 -24529.042,E2 -24529.042} C_VEL
LIN {X 0,Y 163.182,Z 516.78,A -85,B 0,C 180,E1 -24532.204,E2 -24532.204} C_VEL
LIN {X 0,Y 158.241,Z 525.23,A -85,B 0,C 180,E1 -24535.511,E2 -24535.511} C_VEL
LIN {X 0,Y 153.064,Z 533.431,A -85,B 0,C 180,E1 -24539.665,E2 -24539.665} C_VEL
LIN {X 0,Y 152.27,Z 534.677,A -85,B 0,C 180,E1 -24540.432,E2 -24540.432} C_VEL
LIN {X 0,Y 149.835,Z 537.547,A -85,B 0,C 180,E1 -24542.171,E2 -24542.171} C_VEL
LIN {X 0,Y 144.434,Z 541.79,A -85,B 0,C 180,E1 -24544.963,E2 -24544.963} C_VEL
LIN {X 0,Y 139.286,Z 545.458,A -85,B 0,C 180,E1 -24548.057,E2 -24548.057} C_VEL
LIN {X 0,Y 137.323,Z 547.37,A -85,B 0,C 180,E1 -24550.221,E2 -24550.221} C_VEL
LIN {X 0,Y 135.255,Z 550.575,A -85,B 0,C 180,E1 -24554.942,E2 -24554.942} C_VEL
LIN {X 0,Y 133.817,Z 553.265,A -85,B 0,C 180,E1 -24560.935,E2 -24560.935} C_VEL
LIN {X 0,Y 133.326,Z 554.593,A -85,B 0,C 180,E1 -24566.979,E2 -24566.979} C_VEL
LIN {X 0,Y 133.391,Z 554.755,A -85,B 0,C 180,E1 -24570,E2 -24570} C_VEL
LIN {X 0,Y 133.464,Z 554.073,A -85,B 0,C 180,E1 -24576.045,E2 -24576.045} C_VEL
LIN {X 0,Y 134.411,Z 552.048,A -85,B 0,C 180,E1 -24582.072,E2 -24582.072} C_VEL
LIN {X 0,Y 136.388,Z 548.631,A -85,B 0,C 180,E1 -24588.009,E2 -24588.009} C_VEL
LIN {X 0,Y 139.75,Z 543.723,A -85,B 0,C 180,E1 -24593.723,E2 -24593.723} C_VEL
LIN {X 0,Y 143.098,Z 538.743,A -85,B 0,C 180,E1 -24598.028,E2 -24598.028} C_VEL
LIN {X 0,Y 147.656,Z 532.131,A -85,B 0,C 180,E1 -24602.375,E2 -24602.375} C_VEL
LIN {X 0,Y 153.231,Z 523.62,A -85,B 0,C 180,E1 -24606.601,E2 -24606.601} C_VEL
LIN {X 0,Y 158.646,Z 514.738,A -85,B 0,C 180,E1 -24609.966,E2 -24609.966} C_VEL
LIN {X 0,Y 164.568,Z 503.98,A -85,B 0,C 180,E1 -24613.1,E2 -24613.1} C_VEL
LIN {X 0,Y 169.702,Z 493.086,A -85,B 0,C 180,E1 -24615.592,E2 -24615.592} C_VEL
LIN {X 0,Y 174.717,Z 481.157,A -85,B 0,C 180,E1 -24617.657,E2 -24617.657} C_VEL
LIN {X 0,Y 179.367,Z 467.932,A -85,B 0,C 180,E1 -24619.388,E2 -24619.388} C_VEL
LIN {X 0,Y 182.967,Z 455.164,A -85,B 0,C 180,E1 -24620.625,E2 -24620.625} C_VEL
LIN {X 0,Y 185.817,Z 441.592,A -85,B 0,C 180,E1 -24621.593,E2 -24621.593} C_VEL
LIN {X 0,Y 187.945,Z 426.836,A -85,B 0,C 180,E1 -24622.254,E2 -24622.254} C_VEL
LIN {X 0,Y 191.572,Z 380.642,A -85,B 0,C 180,E1 -24623.693,E2 -24623.693} C_VEL
LIN {X 0,Y 191.587,Z 379.322,A -85,B 0,C 180,E1 -24623.769,E2 -24623.769} C_VEL
LIN {X 0,Y 187.796,Z 369.678,A -85,B 0,C 180,E1 -24626.012,E2 -24626.012} C_VEL
LIN {X 0,Y 184.004,Z 361.19,A -85,B 0,C 180,E1 -24628.412,E2 -24628.412} C_VEL
LIN {X 0,Y 181.222,Z 355.801,A -85,B 0,C 180,E1 -24630.286,E2 -24630.286} C_VEL
LIN {X 0,Y 176.374,Z 348.129,A -85,B 0,C 180,E1 -24633.847,E2 -24633.847} C_VEL
LIN {X 0,Y 173.653,Z 344.134,A -85,B 0,C 180,E1 -24636.127,E2 -24636.127} C_VEL
LIN {X 0,Y 171.026,Z 340.367,A -85,B 0,C 180,E1 -24638.611,E2 -24638.611} C_VEL
LIN {X 0,Y 168.431,Z 336.733,A -85,B 0,C 180,E1 -24641.448,E2 -24641.448} C_VEL
LIN {X 0,Y 167.123,Z 335.26,A -85,B 0,C 180,E1 -24643.038,E2 -24643.038} C_VEL
LIN {X 0,Y 164.785,Z 331.546,A -85,B 0,C 180,E1 -24646.591,E2 -24646.591} C_VEL
LIN {X 0,Y 161.07,Z 326.074,A -85,B 0,C 180,E1 -24657.499,E2 -24657.499} C_VEL
LIN {X 0,Y 160.956,Z 325.662,A -85,B 0,C 180,E1 -24660,E2 -24660} C_VEL
LIN {X 0,Y 161.179,Z 326.522,A -85,B 0,C 180,E1 -24663.75,E2 -24663.75} C_VEL
LIN {X 0,Y 164.063,Z 330.926,A -85,B 0,C 180,E1 -24672.368,E2 -24672.368} C_VEL
LIN {X 0,Y 164.833,Z 331.661,A -85,B 0,C 180,E1 -24673.677,E2 -24673.677} C_VEL
LIN {X 0,Y 166.996,Z 335.117,A -85,B 0,C 180,E1 -24676.976,E2 -24676.976} C_VEL
LIN {X 0,Y 168.357,Z 336.626,A -85,B 0,C 180,E1 -24678.639,E2 -24678.639} C_VEL
LIN {X 0,Y 171.151,Z 340.514,A -85,B 0,C 180,E1 -24681.689,E2 -24681.689} C_VEL
LIN {X 0,Y 175.129,Z 346.285,A -85,B 0,C 180,E1 -24685.318,E2 -24685.318} C_VEL
LIN {X 0,Y 179.121,Z 352.309,A -85,B 0,C 180,E1 -24688.408,E2 -24688.408} C_VEL
LIN {X 0,Y 184.546,Z 361.497,A -85,B 0,C 180,E1 -24692.058,E2 -24692.058} C_VEL
LIN {X 0,Y 188.044,Z 368.229,A -85,B 0,C 180,E1 -24694.179,E2 -24694.179} C_VEL
LIN {X 0,Y 191.773,Z 377.434,A -85,B 0,C 180,E1 -24696.367,E2 -24696.367} C_VEL
LIN {X 0,Y 188.173,Z 423.457,A -85,B 0,C 180,E1 -24697.792,E2 -24697.792} C_VEL
LIN {X 0,Y 186.195,Z 438.131,A -85,B 0,C 180,E1 -24698.446,E2 -24698.446} C_VEL
LIN {X 0,Y 183.518,Z 451.417,A -85,B 0,C 180,E1 -24699.368,E2 -24699.368} C_VEL
LIN {X 0,Y 180.247,Z 463.552,A -85,B 0,C 180,E1 -24700.509,E2 -24700.509} C_VEL
LIN {X 0,Y 176.236,Z 475.729,A -85,B 0,C 180,E1 -24702.036,E2 -24702.036} C_VEL
LIN {X 0,Y 171.343,Z 488.137,A -85,B 0,C 180,E1 -24704.079,E2 -24704.079} C_VEL
LIN {X 0,Y 166.131,Z 499.629,A -85,B 0,C 180,E1 -24706.573,E2 -24706.573} C_VEL
LIN {X 0,Y 161.079,Z 509.034,A -85,B 0,C 180,E1 -24709.122,E2 -24709.122} C_VEL
LIN {X 0,Y 155.53,Z 518.486,A -85,B 0,C 180,E1 -24712.409,E2 -24712.409} C_VEL
LIN {X 0,Y 149.704,Z 527.497,A -85,B 0,C 180,E1 -24716.523,E2 -24716.523} C_VEL
LIN {X 0,Y 144.716,Z 534.759,A -85,B 0,C 180,E1 -24720.946,E2 -24720.946} C_VEL
LIN {X 0,Y 141.367,Z 539.839,A -85,B 0,C 180,E1 -24725.003,E2 -24725.003} C_VEL
LIN {X 0,Y 137.524,Z 545.102,A -85,B 0,C 180,E1 -24730.599,E2 -24730.599} C_VEL
LIN {X 0,Y 135.585,Z 548.04,A -85,B 0,C 180,E1 -24734.979,E2 -24734.979} C_VEL
LIN {X 0,Y 134.041,Z 550.733,A -85,B 0,C 180,E1 -24740.95,E2 -24740.95} C_VEL
LIN {X 0,Y 133.404,Z 552.077,A -85,B 0,C 180,E1 -24746.98,E2 -24746.98} C_VEL
LIN {X 0,Y 133.449,Z 552.252,A -85,B 0,C 180,E1 -24750,E2 -24750} C_VEL
LIN {X 0,Y 133.58,Z 551.618,A -85,B 0,C 180,E1 -24756.04,E2 -24756.04} C_VEL
LIN {X 0,Y 134.038,Z 550.801,A -85,B 0,C 180,E1 -24759.05,E2 -24759.05} C_VEL
LIN {X 0,Y 135.564,Z 548.149,A -85,B 0,C 180,E1 -24765.023,E2 -24765.023} C_VEL
LIN {X 0,Y 138.327,Z 544.071,A -85,B 0,C 180,E1 -24770.833,E2 -24770.833} C_VEL
LIN {X 0,Y 141.281,Z 540.036,A -85,B 0,C 180,E1 -24775.013,E2 -24775.013} C_VEL
LIN {X 0,Y 144.715,Z 534.987,A -85,B 0,C 180,E1 -24779.054,E2 -24779.054} C_VEL
LIN {X 0,Y 149.653,Z 527.777,A -85,B 0,C 180,E1 -24783.49,E2 -24783.49} C_VEL
LIN {X 0,Y 155.456,Z 518.855,A -85,B 0,C 180,E1 -24787.611,E2 -24787.611} C_VEL
LIN {X 0,Y 160.989,Z 509.479,A -85,B 0,C 180,E1 -24790.905,E2 -24790.905} C_VEL
LIN {X 0,Y 167.008,Z 498.109,A -85,B 0,C 180,E1 -24793.942,E2 -24793.942} C_VEL
LIN {X 0,Y 172.259,Z 486.351,A -85,B 0,C 180,E1 -24796.399,E2 -24796.399} C_VEL
LIN {X 0,Y 176.712,Z 474.931,A -85,B 0,C 180,E1 -24798.218,E2 -24798.218} C_VEL
LIN {X 0,Y 180.773,Z 462.556,A -85,B 0,C 180,E1 -24799.725,E2 -24799.725} C_VEL
LIN {X 0,Y 184.292,Z 448.819,A -85,B 0,C 180,E1 -24800.985,E2 -24800.985} C_VEL
LIN {X 0,Y 187.011,Z 434.462,A -85,B 0,C 180,E1 -24801.89,E2 -24801.89} C_VEL
LIN {X 0,Y 188.741,Z 419.3,A -85,B 0,C 180,E1 -24802.488,E2 -24802.488} C_VEL
LIN {X 0,Y 192.003,Z 378.161,A -85,B 0,C 180,E1 -24803.713,E2 -24803.713} C_VEL
LIN {X 0,Y 191.59,Z 376.575,A -85,B 0,C 180,E1 -24803.981,E2 -24803.981} C_VEL
LIN {X 0,Y 187.13,Z 366.046,A -85,B 0,C 180,E1 -24806.62,E2 -24806.62} C_VEL
LIN {X 0,Y 181.569,Z 356.191,A -85,B 0,C 180,E1 -24810.15,E2 -24810.15} C_VEL
LIN {X 0,Y 176.686,Z 348.414,A -85,B 0,C 180,E1 -24813.735,E2 -24813.735} C_VEL
LIN {X 0,Y 173.692,Z 344.109,A -85,B 0,C 180,E1 -24816.248,E2 -24816.248} C_VEL
LIN {X 0,Y 171.159,Z 340.467,A -85,B 0,C 180,E1 -24818.667,E2 -24818.667} C_VEL
LIN {X 0,Y 168.499,Z 336.744,A -85,B 0,C 180,E1 -24821.613,E2 -24821.613} C_VEL
LIN {X 0,Y 165.235,Z 332.436,A -85,B 0,C 180,E1 -24826.157,E2 -24826.157} C_VEL
LIN {X 0,Y 164.579,Z 331.204,A -85,B 0,C 180,E1 -24827.358,E2 -24827.358} C_VEL
LIN {X 0,Y 161.278,Z 326.109,A -85,B 0,C 180,E1 -24838.751,E2 -24838.751} C_VEL
LIN {X 0,Y 161.283,Z 326.109,A -85,B 0,C 180,E1 -24841.248,E2 -24841.248} C_VEL
LIN {X 0,Y 164.839,Z 331.521,A -85,B 0,C 180,E1 -24853.013,E2 -24853.013} C_VEL
LIN {X 0,Y 167.118,Z 335.18,A -85,B 0,C 180,E1 -24856.585,E2 -24856.585} C_VEL
LIN {X 0,Y 168.393,Z 336.525,A -85,B 0,C 180,E1 -24858.162,E2 -24858.162} C_VEL
LIN {X 0,Y 170.989,Z 340.289,A -85,B 0,C 180,E1 -24861.078,E2 -24861.078} C_VEL
LIN {X 0,Y 172.099,Z 341.786,A -85,B 0,C 180,E1 -24862.178,E2 -24862.178} C_VEL
LIN {X 0,Y 175.312,Z 346.475,A -85,B 0,C 180,E1 -24865.068,E2 -24865.068} C_VEL
LIN {X 0,Y 178.293,Z 351.031,A -85,B 0,C 180,E1 -24867.432,E2 -24867.432} C_VEL
LIN {X 0,Y 182.573,Z 358.012,A -85,B 0,C 180,E1 -24870.447,E2 -24870.447} C_VEL
LIN {X 0,Y 186.958,Z 367.367,A -85,B 0,C 180,E1 -24873.303,E2 -24873.303} C_VEL
LIN {X 0,Y 190.904,Z 377.097,A -85,B 0,C 180,E1 -24875.681,E2 -24875.681} C_VEL
LIN {X 0,Y 191.859,Z 379.714,A -85,B 0,C 180,E1 -24876.238,E2 -24876.238} C_VEL
LIN {X 0,Y 187.938,Z 428.747,A -85,B 0,C 180,E1 -24877.757,E2 -24877.757} C_VEL
LIN {X 0,Y 185.711,Z 443.391,A -85,B 0,C 180,E1 -24878.476,E2 -24878.476} C_VEL
LIN {X 0,Y 182.62,Z 456.999,A -85,B 0,C 180,E1 -24879.46,E2 -24879.46} C_VEL
LIN {X 0,Y 178.773,Z 470.229,A -85,B 0,C 180,E1 -24880.822,E2 -24880.822} C_VEL
LIN {X 0,Y 174.154,Z 482.987,A -85,B 0,C 180,E1 -24882.569,E2 -24882.569} C_VEL
LIN {X 0,Y 169.203,Z 494.594,A -85,B 0,C 180,E1 -24884.661,E2 -24884.661} C_VEL
LIN {X 0,Y 163.54,Z 506.209,A -85,B 0,C 180,E1 -24887.404,E2 -24887.404} C_VEL
LIN {X 0,Y 157.705,Z 516.595,A -85,B 0,C 180,E1 -24890.578,E2 -24890.578} C_VEL
LIN {X 0,Y 152.43,Z 525.166,A -85,B 0,C 180,E1 -24893.996,E2 -24893.996} C_VEL
LIN {X 0,Y 146.939,Z 533.366,A -85,B 0,C 180,E1 -24898.257,E2 -24898.257} C_VEL
LIN {X 0,Y 142.871,Z 539.304,A -85,B 0,C 180,E1 -24902.306,E2 -24902.306} C_VEL
LIN {X 0,Y 139.778,Z 543.823,A -85,B 0,C 180,E1 -24906.283,E2 -24906.283} C_VEL
LIN {X 0,Y 137.323,Z 547.37,A -85,B 0,C 180,E1 -24910.221,E2 -24910.221} C_VEL
LIN {X 0,Y 135.523,Z 549.103,A -85,B 0,C 180,E1 -24912.47,E2 -24912.47} C_VEL
LIN {X 0,Y 131.249,Z 551.39,A -85,B 0,C 180,E1 -24916.187,E2 -24916.187} C_VEL
LIN {X 0,Y 128.055,Z 552.795,A -85,B 0,C 180,E1 -24919.356,E2 -24919.356} C_VEL
LIN {X 0,Y 126.635,Z 553.605,A -85,B 0,C 180,E1 -24921.922,E2 -24921.922} C_VEL
LIN {X 0,Y 126.465,Z 553.82,A -85,B 0,C 180,E1 -24922.808,E2 -24922.808} C_VEL
LIN {X 0,Y 126.241,Z 554.527,A -85,B 0,C 180,E1 -24926.809,E2 -24926.809} C_VEL
LIN {X 0,Y 126.307,Z 554.689,A -85,B 0,C 180,E1 -24930,E2 -24930} C_VEL
LIN {X 0,Y 126.407,Z 554.006,A -85,B 0,C 180,E1 -24936.384,E2 -24936.384} C_VEL
LIN {X 0,Y 127.438,Z 551.98,A -85,B 0,C 180,E1 -24942.744,E2 -24942.744} C_VEL
LIN {X 0,Y 129.62,Z 548.563,A -85,B 0,C 180,E1 -24948.985,E2 -24948.985} C_VEL
LIN {X 0,Y 133.239,Z 543.654,A -85,B 0,C 180,E1 -24954.959,E2 -24954.959} C_VEL
LIN {X 0,Y 136.686,Z 538.883,A -85,B 0,C 180,E1 -24959.274,E2 -24959.274} C_VEL
LIN {X 0,Y 141.694,Z 532.063,A -85,B 0,C 180,E1 -24963.917,E2 -24963.917} C_VEL
LIN {X 0,Y 147.555,Z 523.55,A -85,B 0,C 180,E1 -24968.256,E2 -24968.256} C_VEL
LIN {X 0,Y 153.241,Z 514.668,A -85,B 0,C 180,E1 -24971.682,E2 -24971.682} C_VEL
LIN {X 0,Y 158.375,Z 505.863,A -85,B 0,C 180,E1 -24974.339,E2 -24974.339} C_VEL
LIN {X 0,Y 164.254,Z 494.19,A -85,B 0,C 180,E1 -24977.115,E2 -24977.115} C_VEL
LIN {X 0,Y 169.401,Z 482.512,A -85,B 0,C 180,E1 -24979.212,E2 -24979.212} C_VEL
LIN {X 0,Y 174.205,Z 469.65,A -85,B 0,C 180,E1 -24980.95,E2 -24980.95} C_VEL
LIN {X 0,Y 178.225,Z 456.266,A -85,B 0,C 180,E1 -24982.29,E2 -24982.29} C_VEL
LIN {X 0,Y 181.339,Z 442.404,A -85,B 0,C 180,E1 -24983.298,E2 -24983.298} C_VEL
LIN {X 0,Y 183.576,Z 427.922,A -85,B 0,C 180,E1 -24983.961,E2 -24983.961} C_VEL
LIN {X 0,Y 187.243,Z 383.243,A -85,B 0,C 180,E1 -24985.359,E2 -24985.359} C_VEL
LIN {X 0,Y 187.196,Z 381.697,A -85,B 0,C 180,E1 -24985.482,E2 -24985.482} C_VEL
LIN {X 0,Y 182.907,Z 370.714,A -85,B 0,C 180,E1 -24988.272,E2 -24988.272} C_VEL
LIN {X 0,Y 178.927,Z 362.13,A -85,B 0,C 180,E1 -24991.078,E2 -24991.078} C_VEL
LIN {X 0,Y 174.334,Z 354.481,A -85,B 0,C 180,E1 -24994.639,E2 -24994.639} C_VEL
LIN {X 0,Y 171.56,Z 350.289,A -85,B 0,C 180,E1 -24997.097,E2 -24997.097} C_VEL
LIN {X 0,Y 169.187,Z 346.778,A -85,B 0,C 180,E1 -24999.483,E2 -24999.483} C_VEL
LIN {X 0,Y 166.387,Z 342.637,A -85,B 0,C 180,E1 -25002.802,E2 -25002.802} C_VEL
LIN {X 0,Y 163.957,Z 339.342,A -85,B 0,C 180,E1 -25006.364,E2 -25006.364} C_VEL
LIN {X 0,Y 163.313,Z 338.057,A -85,B 0,C 180,E1 -25007.575,E2 -25007.575} C_VEL
LIN {X 0,Y 160.668,Z 334.74,A -85,B 0,C 180,E1 -25014.273,E2 -25014.273} C_VEL
LIN {X 0,Y 160.15,Z 332.998,A -85,B 0,C 180,E1 -25018.114,E2 -25018.114} C_VEL
LIN {X 0,Y 160.108,Z 332.839,A -85,B 0,C 180,E1 -25021.258,E2 -25021.258} C_VEL
LIN {X 0,Y 160.415,Z 334.031,A -85,B 0,C 180,E1 -25024.555,E2 -25024.555} C_VEL
LIN {X 0,Y 162.956,Z 337.852,A -85,B 0,C 180,E1 -25031.979,E2 -25031.979} C_VEL
LIN {X 0,Y 163.528,Z 338.447,A -85,B 0,C 180,E1 -25033.012,E2 -25033.012} C_VEL
LIN {X 0,Y 165.69,Z 341.944,A -85,B 0,C 180,E1 -25036.479,E2 -25036.479} C_VEL
LIN {X 0,Y 166.878,Z 343.416,A -85,B 0,C 180,E1 -25038.016,E2 -25038.016} C_VEL
LIN {X 0,Y 170.327,Z 348.442,A -85,B 0,C 180,E1 -25041.877,E2 -25041.877} C_VEL
LIN {X 0,Y 173.127,Z 352.677,A -85,B 0,C 180,E1 -25044.509,E2 -25044.509} C_VEL
LIN {X 0,Y 176.771,Z 358.429,A -85,B 0,C 180,E1 -25047.494,E2 -25047.494} C_VEL
LIN {X 0,Y 181.776,Z 367.228,A -85,B 0,C 180,E1 -25051.065,E2 -25051.065} C_VEL
LIN {X 0,Y 184.92,Z 373.604,A -85,B 0,C 180,E1 -25053.099,E2 -25053.099} C_VEL
LIN {X 0,Y 187.438,Z 380.022,A -85,B 0,C 180,E1 -25054.692,E2 -25054.692} C_VEL
LIN {X 0,Y 184.395,Z 418.394,A -85,B 0,C 180,E1 -25055.881,E2 -25055.881} C_VEL
LIN {X 0,Y 182.688,Z 433.591,A -85,B 0,C 180,E1 -25056.462,E2 -25056.462} C_VEL
LIN {X 0,Y 179.994,Z 447.594,A -85,B 0,C 180,E1 -25057.294,E2 -25057.294} C_VEL
LIN {X 0,Y 176.299,Z 461.638,A -85,B 0,C 180,E1 -25058.527,E2 -25058.527} C_VEL
LIN {X 0,Y 172.131,Z 474.221,A -85,B 0,C 180,E1 -25060.045,E2 -25060.045} C_VEL
LIN {X 0,Y 166.962,Z 487.071,A -85,B 0,C 180,E1 -25062.11,E2 -25062.11} C_VEL
LIN {X 0,Y 161.585,Z 498.631,A -85,B 0,C 180,E1 -25064.586,E2 -25064.586} C_VEL
LIN {X 0,Y 155.775,Z 509.104,A -85,B 0,C 180,E1 -25067.411,E2 -25067.411} C_VEL
LIN {X 0,Y 149.964,Z 518.555,A -85,B 0,C 180,E1 -25070.753,E2 -25070.753} C_VEL
LIN {X 0,Y 143.829,Z 527.566,A -85,B 0,C 180,E1 -25074.961,E2 -25074.961} C_VEL
LIN {X 0,Y 138.537,Z 534.827,A -85,B 0,C 180,E1 -25079.516,E2 -25079.516} C_VEL
LIN {X 0,Y 133.825,Z 541.344,A -85,B 0,C 180,E1 -25085.158,E2 -25085.158} C_VEL
LIN {X 0,Y 130.018,Z 546.231,A -85,B 0,C 180,E1 -25091.076,E2 -25091.076} C_VEL
LIN {X 0,Y 127.69,Z 549.627,A -85,B 0,C 180,E1 -25097.282,E2 -25097.282} C_VEL
LIN {X 0,Y 126.532,Z 551.638,A -85,B 0,C 180,E1 -25103.622,E2 -25103.622} C_VEL
LIN {X 0,Y 126.36,Z 552.319,A -85,B 0,C 180,E1 -25110,E2 -25110} C_VEL
LIN {X 0,Y 126.532,Z 551.684,A -85,B 0,C 180,E1 -25116.378,E2 -25116.378} C_VEL
LIN {X 0,Y 127.68,Z 549.714,A -85,B 0,C 180,E1 -25122.719,E2 -25122.719} C_VEL
LIN {X 0,Y 129.987,Z 546.361,A -85,B 0,C 180,E1 -25128.929,E2 -25128.929} C_VEL
LIN {X 0,Y 133.749,Z 541.524,A -85,B 0,C 180,E1 -25134.857,E2 -25134.857} C_VEL
LIN {X 0,Y 138.247,Z 535.425,A -85,B 0,C 180,E1 -25140.205,E2 -25140.205} C_VEL
LIN {X 0,Y 143.759,Z 527.842,A -85,B 0,C 180,E1 -25145.058,E2 -25145.058} C_VEL
LIN {X 0,Y 149.885,Z 518.919,A -85,B 0,C 180,E1 -25149.271,E2 -25149.271} C_VEL
LIN {X 0,Y 155.682,Z 509.543,A -85,B 0,C 180,E1 -25152.62,E2 -25152.62} C_VEL
LIN {X 0,Y 161.76,Z 498.576,A -85,B 0,C 180,E1 -25155.593,E2 -25155.593} C_VEL
LIN {X 0,Y 167.434,Z 486.413,A -85,B 0,C 180,E1 -25158.161,E2 -25158.161} C_VEL
LIN {X 0,Y 172.058,Z 474.992,A -85,B 0,C 180,E1 -25159.983,E2 -25159.983} C_VEL
LIN {X 0,Y 176.274,Z 462.616,A -85,B 0,C 180,E1 -25161.483,E2 -25161.483} C_VEL
LIN {X 0,Y 179.917,Z 448.877,A -85,B 0,C 180,E1 -25162.738,E2 -25162.738} C_VEL
LIN {X 0,Y 182.724,Z 434.517,A -85,B 0,C 180,E1 -25163.638,E2 -25163.638} C_VEL
LIN {X 0,Y 184.438,Z 420.157,A -85,B 0,C 180,E1 -25164.212,E2 -25164.212} C_VEL
LIN {X 0,Y 187.631,Z 381.454,A -85,B 0,C 180,E1 -25165.357,E2 -25165.357} C_VEL
LIN {X 0,Y 187.532,Z 379.905,A -85,B 0,C 180,E1 -25165.504,E2 -25165.504} C_VEL
LIN {X 0,Y 183.813,Z 370.839,A -85,B 0,C 180,E1 -25167.879,E2 -25167.879} C_VEL
LIN {X 0,Y 178.604,Z 361.42,A -85,B 0,C 180,E1 -25171.421,E2 -25171.421} C_VEL
LIN {X 0,Y 174.316,Z 354.348,A -85,B 0,C 180,E1 -25174.795,E2 -25174.795} C_VEL
LIN {X 0,Y 171.662,Z 350.348,A -85,B 0,C 180,E1 -25177.171,E2 -25177.171} C_VEL
LIN {X 0,Y 169.365,Z 346.906,A -85,B 0,C 180,E1 -25179.505,E2 -25179.505} C_VEL
LIN {X 0,Y 166.812,Z 343.099,A -85,B 0,C 180,E1 -25182.531,E2 -25182.531} C_VEL
LIN {X 0,Y 163.962,Z 339.231,A -85,B 0,C 180,E1 -25186.758,E2 -25186.758} C_VEL
LIN {X 0,Y 163.292,Z 338.051,A -85,B 0,C 180,E1 -25188.046,E2 -25188.046} C_VEL
LIN {X 0,Y 160.398,Z 333.056,A -85,B 0,C 180,E1 -25199.372,E2 -25199.372} C_VEL
LIN {X 0,Y 160.423,Z 333.3,A -85,B 0,C 180,E1 -25201.569,E2 -25201.569} C_VEL
LIN {X 0,Y 163.64,Z 338.485,A -85,B 0,C 180,E1 -25212.518,E2 -25212.518} C_VEL
LIN {X 0,Y 165.959,Z 342.163,A -85,B 0,C 180,E1 -25216.277,E2 -25216.277} C_VEL
LIN {X 0,Y 166.975,Z 343.45,A -85,B 0,C 180,E1 -25217.609,E2 -25217.609} C_VEL
LIN {X 0,Y 170.314,Z 348.279,A -85,B 0,C 180,E1 -25221.404,E2 -25221.404} C_VEL
LIN {X 0,Y 173.224,Z 352.694,A -85,B 0,C 180,E1 -25224.175,E2 -25224.175} C_VEL
LIN {X 0,Y 176.962,Z 358.599,A -85,B 0,C 180,E1 -25227.255,E2 -25227.255} C_VEL
LIN {X 0,Y 180.091,Z 364.254,A -85,B 0,C 180,E1 -25229.576,E2 -25229.576} C_VEL
LIN {X 0,Y 183.676,Z 372.233,A -85,B 0,C 180,E1 -25232.066,E2 -25232.066} C_VEL
LIN {X 0,Y 187.395,Z 381.836,A -85,B 0,C 180,E1 -25234.476,E2 -25234.476} C_VEL
LIN {X 0,Y 187.359,Z 384.717,A -85,B 0,C 180,E1 -25234.651,E2 -25234.651} C_VEL
LIN {X 0,Y 183.511,Z 429.965,A -85,B 0,C 180,E1 -25236.053,E2 -25236.053} C_VEL
LIN {X 0,Y 181.214,Z 444.096,A -85,B 0,C 180,E1 -25236.766,E2 -25236.766} C_VEL
LIN {X 0,Y 177.879,Z 458.069,A -85,B 0,C 180,E1 -25237.797,E2 -25237.797} C_VEL
LIN {X 0,Y 173.618,Z 471.934,A -85,B 0,C 180,E1 -25239.271,E2 -25239.271} C_VEL
LIN {X 0,Y 168.825,Z 484.351,A -85,B 0,C 180,E1 -25241.018,E2 -25241.018} C_VEL
LIN {X 0,Y 163.731,Z 495.706,A -85,B 0,C 180,E1 -25243.14,E2 -25243.14} C_VEL
LIN {X 0,Y 158.358,Z 506.145,A -85,B 0,C 180,E1 -25245.655,E2 -25245.655} C_VEL
LIN {X 0,Y 152.285,Z 516.531,A -85,B 0,C 180,E1 -25248.881,E2 -25248.881} C_VEL
LIN {X 0,Y 146.729,Z 525.101,A -85,B 0,C 180,E1 -25252.361,E2 -25252.361} C_VEL
LIN {X 0,Y 140.929,Z 533.301,A -85,B 0,C 180,E1 -25256.733,E2 -25256.733} C_VEL
LIN {X 0,Y 136.325,Z 539.607,A -85,B 0,C 180,E1 -25261.211,E2 -25261.211} C_VEL
LIN {X 0,Y 132.288,Z 545.147,A -85,B 0,C 180,E1 -25266.519,E2 -25266.519} C_VEL
LIN {X 0,Y 129.616,Z 548.634,A -85,B 0,C 180,E1 -25271.015,E2 -25271.015} C_VEL
LIN {X 0,Y 127.425,Z 552.027,A -85,B 0,C 180,E1 -25277.255,E2 -25277.255} C_VEL
LIN {X 0,Y 126.465,Z 553.82,A -85,B 0,C 180,E1 -25282.808,E2 -25282.808} C_VEL
LIN {X 0,Y 126.015,Z 554.226,A -85,B 0,C 180,E1 -25284.573,E2 -25284.573} C_VEL
LIN {X 0,Y 124.541,Z 554.62,A -85,B 0,C 180,E1 -25287.195,E2 -25287.195} C_VEL
LIN {X 0,Y 120.253,Z 554.526,A -85,B 0,C 180,E1 -25293.45,E2 -25293.45} C_VEL
LIN {X 0,Y 119.371,Z 554.043,A -85,B 0,C 180,E1 -25296.285,E2 -25296.285} C_VEL
LIN {X 0,Y 119.363,Z 553.82,A -85,B 0,C 180,E1 -25297.24,E2 -25297.24} C_VEL
LIN {X 0,Y 120.495,Z 551.913,A -85,B 0,C 180,E1 -25303.492,E2 -25303.492} C_VEL
LIN {X 0,Y 122.901,Z 548.495,A -85,B 0,C 180,E1 -25310.066,E2 -25310.066} C_VEL
LIN {X 0,Y 126.798,Z 543.586,A -85,B 0,C 180,E1 -25316.321,E2 -25316.321} C_VEL
LIN {X 0,Y 130.331,Z 539.033,A -85,B 0,C 180,E1 -25320.636,E2 -25320.636} C_VEL
LIN {X 0,Y 135.826,Z 531.994,A -85,B 0,C 180,E1 -25325.598,E2 -25325.598} C_VEL
LIN {X 0,Y 142.015,Z 523.481,A -85,B 0,C 180,E1 -25330.04,E2 -25330.04} C_VEL
LIN {X 0,Y 148.001,Z 514.599,A -85,B 0,C 180,E1 -25333.514,E2 -25333.514} C_VEL
LIN {X 0,Y 153.352,Z 505.793,A -85,B 0,C 180,E1 -25336.203,E2 -25336.203} C_VEL
LIN {X 0,Y 159.485,Z 494.119,A -85,B 0,C 180,E1 -25338.993,E2 -25338.993} C_VEL
LIN {X 0,Y 164.854,Z 482.441,A -85,B 0,C 180,E1 -25341.079,E2 -25341.079} C_VEL
LIN {X 0,Y 169.818,Z 469.578,A -85,B 0,C 180,E1 -25342.812,E2 -25342.812} C_VEL
LIN {X 0,Y 173.979,Z 456.192,A -85,B 0,C 180,E1 -25344.137,E2 -25344.137} C_VEL
LIN {X 0,Y 177.185,Z 442.327,A -85,B 0,C 180,E1 -25345.14,E2 -25345.14} C_VEL
LIN {X 0,Y 179.462,Z 428.134,A -85,B 0,C 180,E1 -25345.783,E2 -25345.783} C_VEL
LIN {X 0,Y 183.168,Z 384.738,A -85,B 0,C 180,E1 -25347.137,E2 -25347.137} C_VEL
LIN {X 0,Y 179.249,Z 374.339,A -85,B 0,C 180,E1 -25349.926,E2 -25349.926} C_VEL
LIN {X 0,Y 176.07,Z 367.38,A -85,B 0,C 180,E1 -25352.348,E2 -25352.348} C_VEL
LIN {X 0,Y 171.707,Z 359.884,A -85,B 0,C 180,E1 -25356,E2 -25356} C_VEL
LIN {X 0,Y 169.237,Z 356.027,A -85,B 0,C 180,E1 -25358.373,E2 -25358.373} C_VEL
LIN {X 0,Y 167.389,Z 353.175,A -85,B 0,C 180,E1 -25360.374,E2 -25360.374} C_VEL
LIN {X 0,Y 164.842,Z 349.263,A -85,B 0,C 180,E1 -25363.593,E2 -25363.593} C_VEL
LIN {X 0,Y 162.339,Z 345.387,A -85,B 0,C 180,E1 -25367.658,E2 -25367.658} C_VEL
LIN {X 0,Y 161.792,Z 344.669,A -85,B 0,C 180,E1 -25368.728,E2 -25368.728} C_VEL
LIN {X 0,Y 159.283,Z 340.065,A -85,B 0,C 180,E1 -25378.104,E2 -25378.104} C_VEL
LIN {X 0,Y 159.224,Z 339.77,A -85,B 0,C 180,E1 -25380,E2 -25380} C_VEL
LIN {X 0,Y 159.359,Z 340.527,A -85,B 0,C 180,E1 -25383.16,E2 -25383.16} C_VEL
LIN {X 0,Y 161.856,Z 344.779,A -85,B 0,C 180,E1 -25391.585,E2 -25391.585} C_VEL
LIN {X 0,Y 162.497,Z 345.726,A -85,B 0,C 180,E1 -25392.835,E2 -25392.835} C_VEL
LIN {X 0,Y 164.72,Z 349.127,A -85,B 0,C 180,E1 -25396.42,E2 -25396.42} C_VEL
LIN {X 0,Y 168.325,Z 354.551,A -85,B 0,C 180,E1 -25400.837,E2 -25400.837} C_VEL
LIN {X 0,Y 170.977,Z 358.738,A -85,B 0,C 180,E1 -25403.506,E2 -25403.506} C_VEL
LIN {X 0,Y 174.333,Z 364.269,A -85,B 0,C 180,E1 -25406.442,E2 -25406.442} C_VEL
LIN {X 0,Y 179.051,Z 372.911,A -85,B 0,C 180,E1 -25410.03,E2 -25410.03} C_VEL
LIN {X 0,Y 181.764,Z 378.734,A -85,B 0,C 180,E1 -25411.913,E2 -25411.913} C_VEL
LIN {X 0,Y 183.261,Z 382.7,A -85,B 0,C 180,E1 -25412.941,E2 -25412.941} C_VEL
LIN {X 0,Y 181.086,Z 409.499,A -85,B 0,C 180,E1 -25413.785,E2 -25413.785} C_VEL
LIN {X 0,Y 179.03,Z 430.272,A -85,B 0,C 180,E1 -25414.476,E2 -25414.476} C_VEL
LIN {X 0,Y 176.436,Z 444.74,A -85,B 0,C 180,E1 -25415.258,E2 -25415.258} C_VEL
LIN {X 0,Y 172.923,Z 458.587,A -85,B 0,C 180,E1 -25416.369,E2 -25416.369} C_VEL
LIN {X 0,Y 168.886,Z 471.017,A -85,B 0,C 180,E1 -25417.754,E2 -25417.754} C_VEL
LIN {X 0,Y 164.045,Z 483.209,A -85,B 0,C 180,E1 -25419.544,E2 -25419.544} C_VEL
LIN {X 0,Y 158.285,Z 495.612,A -85,B 0,C 180,E1 -25422.003,E2 -25422.003} C_VEL
LIN {X 0,Y 152.796,Z 505.615,A -85,B 0,C 180,E1 -25424.527,E2 -25424.527} C_VEL
LIN {X 0,Y 146.445,Z 515.66,A -85,B 0,C 180,E1 -25427.789,E2 -25427.789} C_VEL
LIN {X 0,Y 140.749,Z 523.997,A -85,B 0,C 180,E1 -25431.38,E2 -25431.38} C_VEL
LIN {X 0,Y 134.713,Z 531.963,A -85,B 0,C 180,E1 -25435.887,E2 -25435.887} C_VEL
LIN {X 0,Y 129.773,Z 538.369,A -85,B 0,C 180,E1 -25440.83,E2 -25440.83} C_VEL
LIN {X 0,Y 126.23,Z 542.811,A -85,B 0,C 180,E1 -25445.319,E2 -25445.319} C_VEL
LIN {X 0,Y 123.289,Z 546.299,A -85,B 0,C 180,E1 -25450,E2 -25450} C_VEL
LIN {X 0,Y 120.758,Z 549.694,A -85,B 0,C 180,E1 -25456.538,E2 -25456.538} C_VEL
LIN {X 0,Y 119.473,Z 551.704,A -85,B 0,C 180,E1 -25463.243,E2 -25463.243} C_VEL
LIN {X 0,Y 119.279,Z 552.385,A -85,B 0,C 180,E1 -25470,E2 -25470} C_VEL
LIN {X 0,Y 119.471,Z 551.75,A -85,B 0,C 180,E1 -25476.756,E2 -25476.756} C_VEL
LIN {X 0,Y 120.749,Z 549.78,A -85,B 0,C 180,E1 -25483.462,E2 -25483.462} C_VEL
LIN {X 0,Y 123.26,Z 546.427,A -85,B 0,C 180,E1 -25490.005,E2 -25490.005} C_VEL
LIN {X 0,Y 127.306,Z 541.59,A -85,B 0,C 180,E1 -25496.208,E2 -25496.208} C_VEL
LIN {X 0,Y 132.422,Z 535.117,A -85,B 0,C 180,E1 -25502.054,E2 -25502.054} C_VEL
LIN {X 0,Y 137.99,Z 527.907,A -85,B 0,C 180,E1 -25506.757,E2 -25506.757} C_VEL
LIN {X 0,Y 144.437,Z 518.984,A -85,B 0,C 180,E1 -25511.061,E2 -25511.061} C_VEL
LIN {X 0,Y 150.526,Z 509.607,A -85,B 0,C 180,E1 -25514.453,E2 -25514.453} C_VEL
LIN {X 0,Y 156.675,Z 498.993,A -85,B 0,C 180,E1 -25517.368,E2 -25517.368} C_VEL
LIN {X 0,Y 162.203,Z 487.763,A -85,B 0,C 180,E1 -25519.787,E2 -25519.787} C_VEL
LIN {X 0,Y 167.575,Z 475.054,A -85,B 0,C 180,E1 -25521.845,E2 -25521.845} C_VEL
LIN {X 0,Y 171.949,Z 462.676,A -85,B 0,C 180,E1 -25523.331,E2 -25523.331} C_VEL
LIN {X 0,Y 175.389,Z 450.235,A -85,B 0,C 180,E1 -25524.48,E2 -25524.48} C_VEL
LIN {X 0,Y 178.292,Z 436.402,A -85,B 0,C 180,E1 -25525.37,E2 -25525.37} C_VEL
LIN {X 0,Y 180.2,Z 421.96,A -85,B 0,C 180,E1 -25525.986,E2 -25525.986} C_VEL
LIN {X 0,Y 183.472,Z 383.861,A -85,B 0,C 180,E1 -25527.117,E2 -25527.117} C_VEL
LIN {X 0,Y 183.406,Z 382.71,A -85,B 0,C 180,E1 -25527.231,E2 -25527.231} C_VEL
LIN {X 0,Y 180.468,Z 375.467,A -85,B 0,C 180,E1 -25529.261,E2 -25529.261} C_VEL
LIN {X 0,Y 176.11,Z 367.271,A -85,B 0,C 180,E1 -25532.44,E2 -25532.44} C_VEL
LIN {X 0,Y 171.937,Z 360.136,A -85,B 0,C 180,E1 -25535.951,E2 -25535.951} C_VEL
LIN {X 0,Y 169.578,Z 356.429,A -85,B 0,C 180,E1 -25538.219,E2 -25538.219} C_VEL
LIN {X 0,Y 167.704,Z 353.461,A -85,B 0,C 180,E1 -25540.252,E2 -25540.252} C_VEL
LIN {X 0,Y 164.836,Z 349.14,A -85,B 0,C 180,E1 -25543.912,E2 -25543.912} C_VEL
LIN {X 0,Y 162.523,Z 345.605,A -85,B 0,C 180,E1 -25547.751,E2 -25547.751} C_VEL
LIN {X 0,Y 162.033,Z 344.853,A -85,B 0,C 180,E1 -25548.744,E2 -25548.744} C_VEL
LIN {X 0,Y 159.533,Z 340.101,A -85,B 0,C 180,E1 -25559.369,E2 -25559.369} C_VEL
LIN {X 0,Y 159.55,Z 340.41,A -85,B 0,C 180,E1 -25561.577,E2 -25561.577} C_VEL
LIN {X 0,Y 162.387,Z 345.242,A -85,B 0,C 180,E1 -25571.863,E2 -25571.863} C_VEL
LIN {X 0,Y 164.71,Z 349.034,A -85,B 0,C 180,E1 -25575.832,E2 -25575.832} C_VEL
LIN {X 0,Y 165.636,Z 350.392,A -85,B 0,C 180,E1 -25577.119,E2 -25577.119} C_VEL
LIN {X 0,Y 168.611,Z 354.866,A -85,B 0,C 180,E1 -25580.67,E2 -25580.67} C_VEL
LIN {X 0,Y 171.371,Z 359.235,A -85,B 0,C 180,E1 -25583.442,E2 -25583.442} C_VEL
LIN {X 0,Y 174.799,Z 364.977,A -85,B 0,C 180,E1 -25586.429,E2 -25586.429} C_VEL
LIN {X 0,Y 177.385,Z 369.863,A -85,B 0,C 180,E1 -25588.469,E2 -25588.469} C_VEL
LIN {X 0,Y 180.801,Z 377.856,A -85,B 0,C 180,E1 -25591.011,E2 -25591.011} C_VEL
LIN {X 0,Y 183.376,Z 384.827,A -85,B 0,C 180,E1 -25592.818,E2 -25592.818} C_VEL
LIN {X 0,Y 179.558,Z 429.127,A -85,B 0,C 180,E1 -25594.2,E2 -25594.2} C_VEL
LIN {X 0,Y 177.222,Z 443.277,A -85,B 0,C 180,E1 -25594.878,E2 -25594.878} C_VEL
LIN {X 0,Y 173.957,Z 456.88,A -85,B 0,C 180,E1 -25595.853,E2 -25595.853} C_VEL
LIN {X 0,Y 169.811,Z 470.107,A -85,B 0,C 180,E1 -25597.185,E2 -25597.185} C_VEL
LIN {X 0,Y 164.866,Z 482.863,A -85,B 0,C 180,E1 -25598.927,E2 -25598.927} C_VEL
LIN {X 0,Y 159.511,Z 494.468,A -85,B 0,C 180,E1 -25601.018,E2 -25601.018} C_VEL
LIN {X 0,Y 153.333,Z 506.081,A -85,B 0,C 180,E1 -25603.79,E2 -25603.79} C_VEL
LIN {X 0,Y 147.006,Z 516.467,A -85,B 0,C 180,E1 -25607.059,E2 -25607.059} C_VEL
LIN {X 0,Y 141.147,Z 525.036,A -85,B 0,C 180,E1 -25610.593,E2 -25610.593} C_VEL
LIN {X 0,Y 135.017,Z 533.235,A -85,B 0,C 180,E1 -25615.071,E2 -25615.071} C_VEL
LIN {X 0,Y 129.797,Z 539.921,A -85,B 0,C 180,E1 -25620.035,E2 -25620.035} C_VEL
LIN {X 0,Y 125.762,Z 545.08,A -85,B 0,C 180,E1 -25625.222,E2 -25625.222} C_VEL
LIN {X 0,Y 122.898,Z 548.568,A -85,B 0,C 180,E1 -25629.934,E2 -25629.934} C_VEL
LIN {X 0,Y 120.484,Z 551.96,A -85,B 0,C 180,E1 -25636.508,E2 -25636.508} C_VEL
LIN {X 0,Y 119.328,Z 553.964,A -85,B 0,C 180,E1 -25643.236,E2 -25643.236} C_VEL
LIN {X 0,Y 119.226,Z 554.622,A -85,B 0,C 180,E1 -25650,E2 -25650} C_VEL
LIN {X 0,Y 119.328,Z 553.939,A -85,B 0,C 180,E1 -25656.765,E2 -25656.765} C_VEL
LIN {X 0,Y 119.363,Z 553.82,A -85,B 0,C 180,E1 -25657.24,E2 -25657.24} C_VEL
LIN {X 0,Y 119.027,Z 553.138,A -85,B 0,C 180,E1 -25660.052,E2 -25660.052} C_VEL
LIN {X 0,Y 117.176,Z 551.533,A -85,B 0,C 180,E1 -25664.721,E2 -25664.721} C_VEL
LIN {X 0,Y 116.072,Z 549.887,A -85,B 0,C 180,E1 -25668.515,E2 -25668.515} C_VEL
LIN {X 0,Y 116.36,Z 548.386,A -85,B 0,C 180,E1 -25671.337,E2 -25671.337} C_VEL
LIN {X 0,Y 116.783,Z 547.806,A -85,B 0,C 180,E1 -25672.245,E2 -25672.245} C_VEL
LIN {X 0,Y 120.439,Z 543.518,A -85,B 0,C 180,E1 -25677.828,E2 -25677.828} C_VEL
LIN {X 0,Y 124.412,Z 538.784,A -85,B 0,C 180,E1 -25682.456,E2 -25682.456} C_VEL
LIN {X 0,Y 130.095,Z 531.925,A -85,B 0,C 180,E1 -25687.426,E2 -25687.426} C_VEL
LIN {X 0,Y 136.62,Z 523.412,A -85,B 0,C 180,E1 -25691.969,E2 -25691.969} C_VEL
LIN {X 0,Y 142.929,Z 514.53,A -85,B 0,C 180,E1 -25695.477,E2 -25695.477} C_VEL
LIN {X 0,Y 149.672,Z 503.77,A -85,B 0,C 180,E1 -25698.702,E2 -25698.702} C_VEL
LIN {X 0,Y 155.507,Z 492.874,A -85,B 0,C 180,E1 -25701.223,E2 -25701.223} C_VEL
LIN {X 0,Y 161.131,Z 480.944,A -85,B 0,C 180,E1 -25703.268,E2 -25703.268} C_VEL
LIN {X 0,Y 166.289,Z 467.714,A -85,B 0,C 180,E1 -25704.969,E2 -25704.969} C_VEL
LIN {X 0,Y 170.584,Z 453.643,A -85,B 0,C 180,E1 -25706.274,E2 -25706.274} C_VEL
LIN {X 0,Y 173.744,Z 439.529,A -85,B 0,C 180,E1 -25707.203,E2 -25707.203} C_VEL
LIN {X 0,Y 175.833,Z 425.638,A -85,B 0,C 180,E1 -25707.777,E2 -25707.777} C_VEL
LIN {X 0,Y 179.197,Z 387.444,A -85,B 0,C 180,E1 -25708.944,E2 -25708.944} C_VEL
LIN {X 0,Y 175.759,Z 378.209,A -85,B 0,C 180,E1 -25711.618,E2 -25711.618} C_VEL
LIN {X 0,Y 173.45,Z 372.95,A -85,B 0,C 180,E1 -25713.532,E2 -25713.532} C_VEL
LIN {X 0,Y 169.755,Z 366.256,A -85,B 0,C 180,E1 -25716.84,E2 -25716.84} C_VEL
LIN {X 0,Y 167.197,Z 362.06,A -85,B 0,C 180,E1 -25719.469,E2 -25719.469} C_VEL
LIN {X 0,Y 165.634,Z 359.561,A -85,B 0,C 180,E1 -25721.284,E2 -25721.284} C_VEL
LIN {X 0,Y 163.229,Z 355.74,A -85,B 0,C 180,E1 -25724.549,E2 -25724.549} C_VEL
LIN {X 0,Y 160.777,Z 351.671,A -85,B 0,C 180,E1 -25728.975,E2 -25728.975} C_VEL
LIN {X 0,Y 158.41,Z 347.176,A -85,B 0,C 180,E1 -25738.093,E2 -25738.093} C_VEL
LIN {X 0,Y 158.357,Z 346.824,A -85,B 0,C 180,E1 -25740,E2 -25740} C_VEL
LIN {X 0,Y 158.439,Z 347.344,A -85,B 0,C 180,E1 -25742.543,E2 -25742.543} C_VEL
LIN {X 0,Y 161.154,Z 352.288,A -85,B 0,C 180,E1 -25751.996,E2 -25751.996} C_VEL
LIN {X 0,Y 163.323,Z 355.837,A -85,B 0,C 180,E1 -25755.762,E2 -25755.762} C_VEL
LIN {X 0,Y 166.644,Z 361.13,A -85,B 0,C 180,E1 -25760.082,E2 -25760.082} C_VEL
LIN {X 0,Y 169.092,Z 365.174,A -85,B 0,C 180,E1 -25762.691,E2 -25762.691} C_VEL
LIN {X 0,Y 172.221,Z 370.605,A -85,B 0,C 180,E1 -25765.594,E2 -25765.594} C_VEL
LIN {X 0,Y 176.479,Z 378.803,A -85,B 0,C 180,E1 -25769.036,E2 -25769.036} C_VEL
LIN {X 0,Y 178.761,Z 384.021,A -85,B 0,C 180,E1 -25770.737,E2 -25770.737} C_VEL
LIN {X 0,Y 179.328,Z 385.642,A -85,B 0,C 180,E1 -25771.165,E2 -25771.165} C_VEL
LIN {X 0,Y 175.461,Z 427.944,A -85,B 0,C 180,E1 -25772.459,E2 -25772.459} C_VEL
LIN {X 0,Y 172.95,Z 442.533,A -85,B 0,C 180,E1 -25773.193,E2 -25773.193} C_VEL
LIN {X 0,Y 169.471,Z 456.403,A -85,B 0,C 180,E1 -25774.229,E2 -25774.229} C_VEL
LIN {X 0,Y 165.278,Z 469.324,A -85,B 0,C 180,E1 -25775.588,E2 -25775.588} C_VEL
LIN {X 0,Y 160.241,Z 481.856,A -85,B 0,C 180,E1 -25777.351,E2 -25777.351} C_VEL
